C03653=1216.229,222.853,-59.172,-177.266,6.356,148.345
C03654=1216.224,223.101,-59.198,-177.264,6.357,148.345
C03655=1216.220,223.350,-59.222,-177.261,6.359,148.345
C03656=1216.216,223.598,-59.248,-177.259,6.362,148.344
C03657=1216.211,223.848,-59.273,-177.256,6.363,148.344
C03658=1216.206,224.096,-59.298,-177.254,6.365,148.344
C03659=1216.202,224.345,-59.323,-177.251,6.367,148.343
C03660=1216.198,224.593,-59.348,-177.248,6.369,148.343
C03661=1216.193,224.843,-59.373,-177.246,6.371,148.343
C03662=1216.188,225.091,-59.398,-177.243,6.373,148.343
C03663=1216.184,225.340,-59.423,-177.240,6.374,148.342
C03664=1216.179,225.589,-59.449,-177.238,6.377,148.342
C03665=1216.175,225.837,-59.473,-177.236,6.379,148.342
C03666=1216.171,226.086,-59.499,-177.233,6.380,148.341
C03667=1216.166,226.334,-59.524,-177.230,6.382,148.341
C03668=1216.162,226.584,-59.549,-177.228,6.384,148.341
C03669=1216.157,226.832,-59.575,-177.225,6.386,148.340
C03670=1216.152,227.081,-59.600,-177.223,6.388,148.340
C03671=1216.147,227.329,-59.625,-177.220,6.390,148.340
C03672=1216.144,227.578,-59.650,-177.218,6.392,148.340
C03673=1216.139,227.827,-59.675,-177.215,6.394,148.339
C03674=1216.134,228.075,-59.701,-177.212,6.396,148.339
C03675=1216.130,228.324,-59.727,-177.210,6.397,148.339
C03676=1216.125,228.572,-59.752,-177.208,6.400,148.339
C03677=1216.121,228.822,-59.777,-177.205,6.401,148.338
C03678=1216.116,229.070,-59.802,-177.202,6.403,148.338
C03679=1216.112,229.318,-59.828,-177.199,6.406,148.338
C03680=1216.107,229.568,-59.853,-177.197,6.408,148.337
C03681=1216.102,229.816,-59.878,-177.194,6.410,148.337
C03682=1216.098,230.065,-59.904,-177.192,6.412,148.337
C03683=1216.093,230.313,-59.930,-177.189,6.414,148.337
C03684=1216.089,230.562,-59.955,-177.187,6.416,148.336
C03685=1216.085,230.811,-59.980,-177.184,6.417,148.336
C03686=1216.080,231.059,-60.006,-177.181,6.419,148.336
C03687=1216.076,231.308,-60.032,-177.179,6.421,148.336
C03688=1216.071,231.557,-60.057,-177.176,6.423,148.335
C03689=1216.067,231.805,-60.083,-177.174,6.425,148.335
C03690=1216.062,232.054,-60.108,-177.171,6.427,148.335
C03691=1216.058,232.303,-60.133,-177.169,6.429,148.334
C03692=1216.053,232.551,-60.159,-177.166,6.431,148.334
C03693=1216.049,232.800,-60.185,-177.164,6.433,148.334
C03694=1216.045,233.049,-60.210,-177.161,6.435,148.334
C03695=1216.040,233.297,-60.236,-177.159,6.437,148.333
C03696=1216.036,233.546,-60.261,-177.156,6.439,148.333
C03697=1216.031,233.795,-60.287,-177.154,6.441,148.333
C03698=1216.026,234.043,-60.313,-177.151,6.443,148.332
C03699=1216.022,234.292,-60.338,-177.149,6.444,148.332
C03700=1216.018,234.540,-60.364,-177.146,6.446,148.332
C03701=1216.012,234.789,-60.390,-177.143,6.448,148.331
C03702=1216.008,235.038,-60.416,-177.141,6.451,148.331
C03703=1216.004,235.286,-60.442,-177.138,6.453,148.331
C03704=1215.999,235.534,-60.467,-177.135,6.455,148.331
C03705=1215.995,235.783,-60.493,-177.133,6.457,148.330
C03706=1215.991,236.032,-60.518,-177.131,6.459,148.330
C03707=1215.986,236.281,-60.544,-177.128,6.461,148.330
C03708=1215.982,236.529,-60.570,-177.125,6.463,148.330
C03709=1215.977,236.778,-60.596,-177.123,6.464,148.329
C03710=1215.972,237.050,-60.624,-177.120,6.466,148.329
C03711=1215.967,237.321,-60.652,-177.117,6.469,148.329
C03712=1215.962,237.592,-60.680,-177.115,6.471,148.329
C03713=1215.957,237.864,-60.708,-177.112,6.473,148.328
C03714=1215.953,238.112,-60.735,-177.110,6.475,148.328
C03715=1215.949,238.361,-60.760,-177.106,6.478,148.328
C03716=1215.944,238.610,-60.787,-177.104,6.479,148.328
C03717=1215.940,238.859,-60.812,-177.102,6.482,148.327
C03718=1215.935,239.107,-60.838,-177.099,6.484,148.327
C03719=1215.931,239.355,-60.864,-177.096,6.485,148.327
C03720=1215.926,239.604,-60.891,-177.094,6.487,148.326
C03721=1215.922,239.853,-60.916,-177.092,6.489,148.326
C03722=1215.917,240.101,-60.942,-177.089,6.491,148.326
C03723=1215.913,240.350,-60.968,-177.086,6.493,148.326
C03724=1215.908,240.599,-60.994,-177.084,6.495,148.326
C03725=1215.904,240.847,-61.020,-177.082,6.497,148.325
C03726=1215.900,241.096,-61.046,-177.079,6.499,148.325
C03727=1215.895,241.345,-61.072,-177.076,6.502,148.325
C03728=1215.890,241.593,-61.098,-177.074,6.504,148.325
C03729=1215.886,241.841,-61.124,-177.071,6.506,148.324
C03730=1215.882,242.090,-61.150,-177.068,6.508,148.324
C03731=1215.877,242.339,-61.176,-177.066,6.510,148.324
C03732=1215.873,242.587,-61.203,-177.064,6.512,148.324
C03733=1215.869,242.836,-61.229,-177.061,6.514,148.323
C03734=1215.863,243.085,-61.255,-177.058,6.515,148.323
C03735=1215.859,243.333,-61.281,-177.056,6.518,148.323
C03736=1215.854,243.582,-61.307,-177.053,6.520,148.323
C03737=1215.850,243.830,-61.334,-177.050,6.522,148.322
C03738=1215.846,244.079,-61.360,-177.048,6.524,148.322
C03739=1215.841,244.328,-61.386,-177.046,6.526,148.322
C03740=1215.837,244.576,-61.412,-177.043,6.528,148.322
C03741=1215.832,244.824,-61.438,-177.040,6.530,148.321
C03742=1215.828,245.073,-61.465,-177.038,6.532,148.321
C03743=1215.823,245.322,-61.491,-177.036,6.534,148.321
C03744=1215.819,245.570,-61.518,-177.033,6.536,148.321
C03745=1215.815,245.819,-61.543,-177.030,6.539,148.320
C03746=1215.810,246.067,-61.570,-177.028,6.541,148.320
C03747=1215.806,246.316,-61.596,-177.025,6.543,148.320
C03748=1215.802,246.564,-61.623,-177.023,6.545,148.320
C03749=1215.797,246.813,-61.649,-177.020,6.547,148.319
C03750=1215.793,247.062,-61.676,-177.018,6.549,148.319
C03751=1215.788,247.311,-61.702,-177.016,6.551,148.319
C03752=1215.783,247.558,-61.728,-177.013,6.553,148.319
C03753=1215.778,247.807,-61.754,-177.010,6.555,148.318
C03754=1215.774,248.055,-61.781,-177.008,6.557,148.318
C03755=1215.770,248.305,-61.807,-177.005,6.559,148.318
C03756=1215.766,248.553,-61.834,-177.002,6.561,148.318
C03757=1215.761,248.801,-61.861,-177.000,6.563,148.318
C03758=1215.757,249.050,-61.886,-176.998,6.565,148.317
C03759=1215.752,249.299,-61.913,-176.995,6.567,148.317
C03760=1215.747,249.547,-61.941,-176.992,6.570,148.317
C03761=1215.743,249.796,-61.966,-176.990,6.572,148.317
C03762=1215.739,250.044,-61.993,-176.987,6.574,148.316
C03763=1215.735,250.293,-62.020,-176.985,6.576,148.316
C03764=1215.730,250.542,-62.046,-176.982,6.578,148.316
C03765=1215.726,250.790,-62.073,-176.980,6.580,148.316
C03766=1215.721,251.038,-62.100,-176.978,6.582,148.316
C03767=1215.716,251.287,-62.126,-176.974,6.585,148.315
C03768=1215.712,251.536,-62.152,-176.972,6.587,148.315
C03769=1215.708,251.784,-62.180,-176.970,6.589,148.315
C03770=1215.704,252.032,-62.206,-176.967,6.591,148.315
C03771=1215.699,252.281,-62.232,-176.965,6.593,148.315
C03772=1215.694,252.530,-62.259,-176.962,6.595,148.314
C03773=1215.690,252.778,-62.286,-176.959,6.597,148.314
C03774=1215.685,253.027,-62.313,-176.957,6.600,148.314
C03775=1215.681,253.275,-62.340,-176.954,6.601,148.314
C03776=1215.677,253.524,-62.366,-176.952,6.603,148.313
C03777=1215.672,253.772,-62.393,-176.950,6.605,148.313
C03778=1215.667,254.021,-62.420,-176.947,6.607,148.313
C03779=1215.663,254.269,-62.446,-176.944,6.610,148.313
C03780=1215.659,254.518,-62.473,-176.942,6.612,148.312
C03781=1215.654,254.766,-62.500,-176.939,6.614,148.312
C03782=1215.650,255.014,-62.527,-176.937,6.616,148.312
C03783=1215.646,255.263,-62.554,-176.934,6.618,148.312
C03784=1215.641,255.512,-62.581,-176.932,6.621,148.312
C03785=1215.636,255.761,-62.608,-176.929,6.623,148.311
C03786=1215.632,256.009,-62.634,-176.926,6.625,148.311
C03787=1215.628,256.258,-62.661,-176.924,6.627,148.311
C03788=1215.623,256.506,-62.688,-176.922,6.629,148.311
C03789=1215.619,256.755,-62.715,-176.919,6.632,148.311
C03790=1215.615,257.003,-62.742,-176.916,6.634,148.310
C03791=1215.610,257.251,-62.769,-176.914,6.636,148.310
C03792=1215.605,257.500,-62.796,-176.912,6.638,148.310
C03793=1215.601,257.749,-62.823,-176.909,6.640,148.310
C03794=1215.597,257.998,-62.850,-176.906,6.643,148.310
C03795=1215.593,258.246,-62.877,-176.904,6.645,148.309
C03796=1215.588,258.494,-62.904,-176.901,6.647,148.309
C03797=1215.584,258.742,-62.932,-176.899,6.649,148.309
C03798=1215.579,258.991,-62.959,-176.896,6.651,148.309
C03799=1215.574,259.239,-62.986,-176.894,6.654,148.309
C03800=1215.570,259.487,-63.012,-176.891,6.656,148.308
C03801=1215.566,259.737,-63.040,-176.889,6.658,148.308
C03802=1215.562,259.985,-63.067,-176.886,6.660,148.308
C03803=1215.557,260.234,-63.094,-176.884,6.661,148.308
C03804=1215.552,260.482,-63.121,-176.881,6.665,148.308
C03805=1215.548,260.731,-63.148,-176.878,6.666,148.307
C03806=1215.543,260.978,-63.176,-176.876,6.669,148.307
C03807=1215.539,261.228,-63.203,-176.874,6.670,148.307
C03808=1215.535,261.476,-63.230,-176.871,6.673,148.307
C03809=1215.531,261.724,-63.257,-176.868,6.675,148.307
C03810=1215.526,261.973,-63.284,-176.866,6.678,148.306
C03811=1215.522,262.221,-63.312,-176.864,6.679,148.306
C03812=1215.518,262.470,-63.339,-176.861,6.682,148.306
C03813=1215.513,262.718,-63.366,-176.858,6.684,148.306
C03814=1215.508,262.991,-63.396,-176.856,6.686,148.306
C03815=1215.503,263.263,-63.426,-176.853,6.689,148.305
C03816=1215.498,263.536,-63.456,-176.850,6.691,148.305
C03817=1215.494,263.809,-63.487,-176.847,6.694,148.305
C03818=1215.489,264.057,-63.514,-176.845,6.696,148.305
C03819=1215.485,264.306,-63.541,-176.842,6.698,148.305
C03820=1215.480,264.554,-63.568,-176.840,6.701,148.305
C03821=1215.476,264.803,-63.596,-176.837,6.703,148.304
C03822=1215.472,265.051,-63.623,-176.835,6.705,148.304
C03823=1215.467,265.299,-63.651,-176.832,6.707,148.304
C03824=1215.463,265.548,-63.678,-176.830,6.710,148.304
C03825=1215.459,265.797,-63.705,-176.827,6.712,148.303
C03826=1215.454,266.045,-63.733,-176.825,6.714,148.303
C03827=1215.450,266.293,-63.760,-176.822,6.716,148.303
C03828=1215.445,266.541,-63.788,-176.820,6.719,148.303
C03829=1215.440,266.791,-63.816,-176.817,6.721,148.303
C03830=1215.436,267.039,-63.844,-176.815,6.723,148.303
C03831=1215.431,267.287,-63.871,-176.812,6.725,148.302
C03832=1215.428,267.536,-63.899,-176.810,6.728,148.302
C03833=1215.423,267.784,-63.926,-176.807,6.730,148.302
C03834=1215.419,268.032,-63.954,-176.805,6.732,148.302
C03835=1215.414,268.281,-63.981,-176.802,6.734,148.302
C03836=1215.410,268.529,-64.009,-176.800,6.737,148.302
C03837=1215.406,268.778,-64.036,-176.797,6.739,148.301
C03838=1215.401,269.026,-64.064,-176.795,6.741,148.301
C03839=1215.396,269.275,-64.092,-176.792,6.744,148.301
C03840=1215.392,269.523,-64.120,-176.790,6.746,148.301
C03841=1215.387,269.771,-64.147,-176.787,6.748,148.301
C03842=1215.384,270.020,-64.175,-176.785,6.750,148.301
C03843=1215.379,270.268,-64.202,-176.782,6.753,148.300
C03844=1215.374,270.517,-64.230,-176.780,6.755,148.300
C03845=1215.370,270.765,-64.258,-176.777,6.757,148.300
C03846=1215.366,271.014,-64.285,-176.774,6.760,148.300
C03847=1215.362,271.262,-64.313,-176.772,6.762,148.300
C03848=1215.357,271.510,-64.341,-176.769,6.764,148.300
C03849=1215.352,271.759,-64.369,-176.767,6.766,148.299
C03850=1215.348,272.008,-64.397,-176.764,6.769,148.299
C03851=1215.344,272.255,-64.425,-176.762,6.771,148.299
C03852=1215.340,272.503,-64.453,-176.759,6.773,148.299
C03853=1215.335,272.753,-64.481,-176.757,6.776,148.299
C03854=1215.330,273.001,-64.508,-176.755,6.778,148.299
C03855=1215.327,273.249,-64.537,-176.752,6.780,148.298
C03856=1215.322,273.498,-64.564,-176.750,6.782,148.298
C03857=1215.318,273.747,-64.592,-176.747,6.785,148.298
C03858=1215.313,273.995,-64.620,-176.745,6.787,148.298
C03859=1215.309,274.242,-64.648,-176.742,6.789,148.298
C03860=1215.305,274.491,-64.676,-176.739,6.792,148.298
C03861=1215.300,274.740,-64.704,-176.737,6.794,148.298
C03862=1215.296,274.988,-64.732,-176.735,6.796,148.297
C03863=1215.292,275.236,-64.760,-176.732,6.799,148.297
C03864=1215.287,275.485,-64.788,-176.729,6.801,148.297
C03865=1215.283,275.733,-64.816,-176.727,6.803,148.297
C03866=1215.278,275.981,-64.844,-176.724,6.806,148.297
C03867=1215.274,276.230,-64.873,-176.722,6.808,148.297
C03868=1215.269,276.478,-64.900,-176.720,6.810,148.297
C03869=1215.265,276.727,-64.928,-176.717,6.813,148.296
C03870=1215.260,276.975,-64.956,-176.714,6.815,148.296
C03871=1215.257,277.224,-64.984,-176.712,6.817,148.296
C03872=1215.252,277.472,-65.013,-176.709,6.820,148.296
C03873=1215.248,277.720,-65.041,-176.707,6.822,148.296
C03874=1215.243,277.969,-65.069,-176.704,6.824,148.296
C03875=1215.239,278.217,-65.097,-176.702,6.827,148.296
C03876=1215.235,278.465,-65.125,-176.700,6.829,148.295
C03877=1215.230,278.714,-65.154,-176.697,6.831,148.295
C03878=1215.226,278.962,-65.182,-176.694,6.834,148.295
C03879=1215.221,279.211,-65.210,-176.692,6.836,148.295
C03880=1215.217,279.459,-65.238,-176.690,6.838,148.295
C03881=1215.213,279.707,-65.267,-176.687,6.841,148.295
C03882=1215.208,279.955,-65.295,-176.685,6.843,148.295
C03883=1215.204,280.204,-65.323,-176.682,6.845,148.294
C03884=1215.200,280.453,-65.352,-176.680,6.848,148.294
C03885=1215.196,280.700,-65.380,-176.677,6.851,148.294
C03886=1215.191,280.949,-65.409,-176.675,6.852,148.294
C03887=1215.187,281.197,-65.437,-176.672,6.856,148.294
C03888=1215.183,281.446,-65.465,-176.670,6.858,148.294
C03889=1215.177,281.694,-65.494,-176.667,6.860,148.294
C03890=1215.174,281.942,-65.522,-176.665,6.863,148.294
C03891=1215.169,282.191,-65.550,-176.663,6.865,148.294
C03892=1215.165,282.439,-65.579,-176.660,6.867,148.293
C03893=1215.161,282.688,-65.608,-176.657,6.870,148.293
C03894=1215.156,282.935,-65.636,-176.655,6.872,148.293
C03895=1215.152,283.184,-65.664,-176.652,6.875,148.293
C03896=1215.148,283.432,-65.692,-176.650,6.877,148.293
C03897=1215.143,283.680,-65.722,-176.648,6.879,148.293
C03898=1215.139,283.929,-65.750,-176.645,6.882,148.293
C03899=1215.135,284.177,-65.778,-176.642,6.884,148.292
C03900=1215.130,284.426,-65.807,-176.640,6.886,148.292
C03901=1215.125,284.674,-65.836,-176.637,6.889,148.292
C03902=1215.121,284.922,-65.864,-176.635,6.891,148.292
C03903=1215.117,285.171,-65.893,-176.633,6.893,148.292
C03904=1215.113,285.418,-65.921,-176.630,6.896,148.292
C03905=1215.108,285.667,-65.950,-176.628,6.898,148.292
C03906=1215.104,285.916,-65.979,-176.625,6.901,148.292
C03907=1215.100,286.163,-66.007,-176.623,6.903,148.292
C03908=1215.095,286.412,-66.036,-176.620,6.905,148.291
C03909=1215.090,286.660,-66.064,-176.618,6.908,148.291
C03910=1215.087,286.908,-66.093,-176.615,6.911,148.291
C03911=1215.082,287.157,-66.122,-176.613,6.914,148.291
C03912=1215.078,287.405,-66.151,-176.610,6.915,148.291
C03913=1215.073,287.654,-66.180,-176.608,6.918,148.291
C03914=1215.069,287.902,-66.208,-176.605,6.921,148.291
C03915=1215.065,288.151,-66.237,-176.603,6.923,148.291
C03916=1215.060,288.399,-66.266,-176.601,6.925,148.290
C03917=1215.057,288.647,-66.295,-176.598,6.928,148.290
C03918=1215.051,288.921,-66.327,-176.595,6.931,148.290
C03919=1215.046,289.196,-66.358,-176.593,6.933,148.290
C03920=1215.042,289.470,-66.391,-176.590,6.936,148.290
C03921=1215.037,289.744,-66.422,-176.587,6.939,148.290
C03922=1215.033,289.993,-66.451,-176.585,6.941,148.290
C03923=1215.029,290.240,-66.480,-176.582,6.944,148.290
C03924=1215.024,290.488,-66.509,-176.580,6.946,148.290
C03925=1215.020,290.737,-66.538,-176.578,6.948,148.290
C03926=1215.015,290.985,-66.567,-176.575,6.951,148.290
C03927=1215.011,291.234,-66.596,-176.573,6.953,148.289
C03928=1215.007,291.482,-66.625,-176.570,6.956,148.289
C03929=1215.003,291.730,-66.653,-176.568,6.958,148.289
C03930=1214.998,291.978,-66.682,-176.565,6.961,148.289
C03931=1214.994,292.226,-66.712,-176.563,6.964,148.289
C03932=1214.989,292.475,-66.741,-176.560,6.965,148.289
C03933=1214.985,292.723,-66.770,-176.558,6.968,148.289
C03934=1214.981,292.972,-66.800,-176.556,6.971,148.289
C03935=1214.976,293.220,-66.827,-176.553,6.974,148.289
C03936=1214.972,293.468,-66.857,-176.551,6.976,148.289
C03937=1214.968,293.716,-66.886,-176.548,6.978,148.288
C03938=1214.964,293.964,-66.916,-176.545,6.981,148.288
C03939=1214.959,294.213,-66.944,-176.543,6.983,148.288
C03940=1214.955,294.461,-66.973,-176.541,6.986,148.288
C03941=1214.950,294.709,-67.003,-176.539,6.988,148.288
C03942=1214.946,294.957,-67.032,-176.536,6.991,148.288
C03943=1214.942,295.206,-67.061,-176.533,6.993,148.288
C03944=1214.938,295.455,-67.091,-176.531,6.995,148.288
C03945=1214.933,295.702,-67.120,-176.528,6.998,148.288
C03946=1214.929,295.950,-67.149,-176.526,7.001,148.288
C03947=1214.924,296.199,-67.179,-176.524,7.004,148.288
C03948=1214.920,296.447,-67.208,-176.522,7.006,148.288
C03949=1214.916,296.696,-67.237,-176.519,7.009,148.288
C03950=1214.912,296.944,-67.266,-176.516,7.011,148.288
C03951=1214.907,297.192,-67.295,-176.514,7.013,148.287
C03952=1214.903,297.440,-67.325,-176.511,7.016,148.287
C03953=1214.898,297.688,-67.354,-176.509,7.018,148.287
C03954=1214.894,297.936,-67.384,-176.507,7.021,148.287
C03955=1214.890,298.185,-67.413,-176.505,7.024,148.287
C03956=1214.886,298.433,-67.443,-176.502,7.027,148.287
C03957=1214.882,298.681,-67.472,-176.500,7.029,148.287
C03958=1214.878,298.930,-67.501,-176.497,7.032,148.287
C03959=1214.873,299.177,-67.531,-176.495,7.034,148.287
C03960=1214.869,299.425,-67.560,-176.492,7.036,148.287
C03961=1214.864,299.674,-67.589,-176.490,7.039,148.287
C03962=1214.860,299.922,-67.619,-176.488,7.041,148.287
C03963=1214.856,300.170,-67.648,-176.485,7.044,148.287
C03964=1214.852,300.418,-67.678,-176.483,7.046,148.287
C03965=1214.848,300.667,-67.707,-176.480,7.049,148.287
C03966=1214.843,300.915,-67.737,-176.478,7.052,148.287
C03967=1214.839,301.164,-67.767,-176.475,7.055,148.287
C03968=1214.834,301.412,-67.796,-176.473,7.057,148.287
C03969=1214.830,301.660,-67.826,-176.471,7.060,148.287
C03970=1214.825,301.908,-67.855,-176.468,7.062,148.287
C03971=1214.821,302.156,-67.884,-176.466,7.064,148.286
C03972=1214.817,302.404,-67.914,-176.464,7.067,148.286
C03973=1214.812,302.652,-67.944,-176.461,7.070,148.286
C03974=1214.808,302.900,-67.974,-176.459,7.073,148.286
C03975=1214.804,303.149,-68.003,-176.457,7.075,148.286
C03976=1214.800,303.397,-68.033,-176.454,7.078,148.286
C03977=1214.796,303.645,-68.062,-176.451,7.080,148.286
C03978=1214.791,303.894,-68.092,-176.449,7.083,148.286
C03979=1214.787,304.141,-68.122,-176.447,7.085,148.286
C03980=1214.783,304.390,-68.152,-176.444,7.088,148.286
C03981=1214.779,304.638,-68.181,-176.442,7.090,148.286
C03982=1214.774,304.887,-68.211,-176.439,7.093,148.286
C03983=1214.770,305.134,-68.242,-176.437,7.095,148.286
C03984=1214.766,305.382,-68.271,-176.435,7.098,148.286
C03985=1214.761,305.631,-68.301,-176.432,7.101,148.286
C03986=1214.757,305.879,-68.331,-176.430,7.103,148.286
C03987=1214.753,306.127,-68.361,-176.427,7.106,148.286
C03988=1214.748,306.375,-68.390,-176.425,7.108,148.286
C03989=1214.744,306.624,-68.420,-176.423,7.112,148.286
C03990=1214.740,306.871,-68.450,-176.421,7.114,148.286
C03991=1214.735,307.120,-68.480,-176.418,7.117,148.286
C03992=1214.731,307.368,-68.511,-176.416,7.119,148.286
C03993=1214.727,307.616,-68.540,-176.414,7.122,148.286
C03994=1214.723,307.864,-68.570,-176.411,7.124,148.286
C03995=1214.718,308.112,-68.600,-176.409,7.127,148.286
C03996=1214.714,308.360,-68.630,-176.407,7.129,148.286
C03997=1214.710,308.608,-68.660,-176.404,7.133,148.286
C03998=1214.706,308.857,-68.690,-176.402,7.135,148.286
C03999=1214.701,309.106,-68.720,-176.399,7.138,148.286
C04000=1214.697,309.353,-68.750,-176.397,7.140,148.285
C04001=1214.693,309.602,-68.780,-176.394,7.143,148.285
C04002=1214.689,309.849,-68.810,-176.392,7.145,148.285
C04003=1214.684,310.098,-68.840,-176.390,7.148,148.285
C04004=1214.680,310.346,-68.870,-176.387,7.150,148.285
C04005=1214.676,310.594,-68.900,-176.385,7.154,148.286
C04006=1214.671,310.842,-68.931,-176.383,7.156,148.286
C04007=1214.667,311.090,-68.960,-176.381,7.159,148.286
C04008=1214.662,311.338,-68.991,-176.378,7.161,148.285
C04009=1214.659,311.587,-69.021,-176.376,7.164,148.285
C04010=1214.654,311.835,-69.051,-176.374,7.167,148.285
C04011=1214.650,312.083,-69.082,-176.371,7.170,148.285
C04012=1214.645,312.331,-69.112,-176.369,7.172,148.285
C04013=1214.641,312.579,-69.142,-176.367,7.174,148.286
C04014=1214.637,312.827,-69.173,-176.364,7.177,148.286
C04015=1214.633,313.075,-69.202,-176.362,7.180,148.285
C04016=1214.629,313.324,-69.233,-176.360,7.183,148.285
C04017=1214.625,313.571,-69.263,-176.358,7.185,148.285
C04018=1214.620,313.820,-69.293,-176.355,7.188,148.285
C04019=1214.616,314.068,-69.324,-176.353,7.190,148.285
C04020=1214.611,314.316,-69.354,-176.351,7.193,148.286
C04021=1214.607,314.564,-69.384,-176.348,7.196,148.286
C04022=1214.602,314.840,-69.418,-176.346,7.199,148.286
C04023=1214.597,315.116,-69.452,-176.343,7.202,148.286
C04024=1214.593,315.392,-69.486,-176.340,7.205,148.286
C04025=1214.588,315.667,-69.520,-176.338,7.208,148.286
C04026=1214.584,315.917,-69.550,-176.335,7.211,148.286
C04027=1214.580,316.164,-69.580,-176.333,7.213,148.286
C04028=1214.576,316.412,-69.611,-176.331,7.216,148.286
C04029=1214.571,316.660,-69.642,-176.329,7.219,148.286
C04030=1214.567,316.908,-69.672,-176.326,7.222,148.286
C04031=1214.563,317.157,-69.702,-176.324,7.224,148.286
C04032=1214.558,317.405,-69.733,-176.322,7.227,148.286
C04033=1214.554,317.653,-69.763,-176.320,7.229,148.286
C04034=1214.550,317.901,-69.794,-176.317,7.232,148.286
C04035=1214.546,318.149,-69.824,-176.315,7.235,148.286
C04036=1214.542,318.397,-69.855,-176.313,7.238,148.286
C04037=1214.537,318.645,-69.886,-176.311,7.240,148.286
C04038=1214.533,318.893,-69.916,-176.308,7.243,148.286
C04039=1214.529,319.141,-69.947,-176.306,7.245,148.286
C04040=1214.525,319.389,-69.978,-176.304,7.249,148.286
C04041=1214.520,319.637,-70.009,-176.301,7.251,148.286
C04042=1214.516,319.885,-70.038,-176.299,7.254,148.286
C04043=1214.512,320.134,-70.069,-176.297,7.257,148.286
C04044=1214.507,320.382,-70.100,-176.294,7.260,148.286
C04045=1214.503,320.630,-70.130,-176.292,7.262,148.286
C04046=1214.499,320.878,-70.161,-176.290,7.265,148.286
C04047=1214.495,321.126,-70.193,-176.288,7.267,148.286
C04048=1214.491,321.374,-70.224,-176.285,7.270,148.286
C04049=1214.487,321.621,-70.254,-176.283,7.273,148.286
C04050=1214.483,321.870,-70.285,-176.281,7.276,148.286
C04051=1214.478,322.118,-70.316,-176.279,7.278,148.286
C04052=1214.473,322.366,-70.347,-176.276,7.281,148.286
C04053=1214.470,322.614,-70.377,-176.275,7.284,148.287
C04054=1214.466,322.862,-70.408,-176.272,7.287,148.287
C04055=1214.461,323.110,-70.439,-176.270,7.289,148.286
C04056=1214.457,323.359,-70.470,-176.268,7.292,148.287
C04057=1214.452,323.607,-70.500,-176.265,7.295,148.287
C04058=1214.449,323.854,-70.531,-176.263,7.298,148.287
C04059=1214.445,324.102,-70.563,-176.261,7.300,148.287
C04060=1214.440,324.350,-70.593,-176.258,7.303,148.287
C04061=1214.435,324.598,-70.624,-176.257,7.306,148.287
C04062=1214.431,324.847,-70.655,-176.254,7.309,148.287
C04063=1214.427,325.094,-70.687,-176.252,7.311,148.287
C04064=1214.423,325.343,-70.718,-176.250,7.314,148.287
C04065=1214.419,325.591,-70.748,-176.248,7.317,148.287
C04066=1214.415,325.839,-70.779,-176.246,7.320,148.287
C04067=1214.411,326.087,-70.811,-176.243,7.322,148.287
C04068=1214.406,326.335,-70.841,-176.241,7.325,148.288
C04069=1214.402,326.583,-70.872,-176.239,7.328,148.287
C04070=1214.398,326.831,-70.903,-176.236,7.331,148.287
C04071=1214.393,327.079,-70.935,-176.235,7.333,148.288
C04072=1214.389,327.327,-70.966,-176.232,7.336,148.288
C04073=1214.385,327.575,-70.997,-176.230,7.339,148.288
C04074=1214.381,327.823,-71.028,-176.228,7.342,148.288
C04075=1214.376,328.071,-71.059,-176.226,7.344,148.288
C04076=1214.372,328.319,-71.090,-176.224,7.347,148.288
C04077=1214.368,328.567,-71.122,-176.222,7.350,148.288
C04078=1214.364,328.815,-71.153,-176.219,7.353,148.288
C04079=1214.361,329.063,-71.184,-176.217,7.356,148.288
C04080=1214.356,329.311,-71.215,-176.215,7.358,148.288
C04081=1214.352,329.560,-71.246,-176.213,7.362,148.289
C04082=1214.348,329.807,-71.277,-176.211,7.364,148.289
C04083=1214.343,330.056,-71.309,-176.208,7.367,148.289
C04084=1214.339,330.303,-71.340,-176.206,7.370,148.289
C04085=1214.334,330.551,-71.371,-176.204,7.373,148.289
C04086=1214.330,330.799,-71.403,-176.202,7.375,148.289
C04087=1214.326,331.047,-71.434,-176.200,7.379,148.289
C04088=1214.322,331.295,-71.466,-176.198,7.381,148.289
C04089=1214.317,331.543,-71.496,-176.195,7.384,148.289
C04090=1214.314,331.791,-71.528,-176.193,7.386,148.289
C04091=1214.309,332.039,-71.559,-176.191,7.390,148.289
C04092=1214.305,332.287,-71.591,-176.189,7.392,148.290
C04093=1214.301,332.535,-71.622,-176.187,7.395,148.290
C04094=1214.297,332.783,-71.653,-176.185,7.398,148.290
C04095=1214.293,333.030,-71.685,-176.183,7.401,148.290
C04096=1214.289,333.279,-71.716,-176.181,7.403,148.290
C04097=1214.284,333.527,-71.748,-176.178,7.406,148.290
C04098=1214.280,333.775,-71.779,-176.177,7.409,148.290
C04099=1214.275,334.023,-71.811,-176.174,7.412,148.290
C04100=1214.272,334.271,-71.843,-176.172,7.414,148.290
C04101=1214.267,334.519,-71.873,-176.170,7.418,148.291
C04102=1214.263,334.767,-71.905,-176.168,7.420,148.291
C04103=1214.260,335.015,-71.937,-176.166,7.423,148.291
C04104=1214.254,335.263,-71.968,-176.164,7.426,148.291
C04105=1214.250,335.511,-72.000,-176.162,7.429,148.291
C04106=1214.246,335.759,-72.032,-176.160,7.431,148.291
C04107=1214.242,336.007,-72.064,-176.158,7.435,148.291
C04108=1214.238,336.255,-72.094,-176.156,7.437,148.292
C04109=1214.233,336.503,-72.127,-176.153,7.440,148.292
C04110=1214.229,336.750,-72.158,-176.152,7.443,148.292
C04111=1214.225,336.998,-72.190,-176.149,7.446,148.292
C04112=1214.221,337.247,-72.221,-176.147,7.448,148.292
C04113=1214.217,337.494,-72.253,-176.145,7.452,148.292
C04114=1214.213,337.743,-72.285,-176.143,7.454,148.292
C04115=1214.208,337.990,-72.317,-176.141,7.457,148.292
C04116=1214.205,338.238,-72.348,-176.139,7.460,148.292
C04117=1214.201,338.487,-72.380,-176.137,7.463,148.293
C04118=1214.196,338.734,-72.412,-176.135,7.466,148.293
C04119=1214.192,338.982,-72.444,-176.133,7.469,148.293
C04120=1214.188,339.230,-72.475,-176.131,7.471,148.293
C04121=1214.183,339.478,-72.507,-176.129,7.475,148.293
C04122=1214.179,339.726,-72.539,-176.127,7.477,148.293
C04123=1214.175,339.973,-72.571,-176.124,7.480,148.293
C04124=1214.171,340.221,-72.603,-176.123,7.483,148.294
C04125=1214.167,340.470,-72.635,-176.121,7.486,148.294
C04126=1214.162,340.748,-72.670,-176.118,7.489,148.294
C04127=1214.157,341.026,-72.706,-176.117,7.492,148.294
C04128=1214.153,341.303,-72.742,-176.114,7.495,148.294
C04129=1214.148,341.582,-72.777,-176.112,7.498,148.295
C04130=1214.144,341.830,-72.809,-176.110,7.502,148.295
C04131=1214.139,342.078,-72.842,-176.108,7.504,148.295
C04132=1214.135,342.325,-72.873,-176.106,7.508,148.295
C04133=1214.131,342.574,-72.905,-176.104,7.510,148.295
C04134=1214.127,342.821,-72.938,-176.102,7.513,148.295
C04135=1214.123,343.069,-72.969,-176.100,7.516,148.296
C04136=1214.119,343.317,-73.002,-176.098,7.519,148.296
C04137=1214.115,343.565,-73.034,-176.096,7.522,148.296
C04138=1214.110,343.813,-73.066,-176.094,7.525,148.296
C04139=1214.106,344.061,-73.098,-176.092,7.527,148.296
C04140=1214.102,344.309,-73.130,-176.090,7.531,148.297
C04141=1214.097,344.556,-73.162,-176.088,7.533,148.297
C04142=1214.094,344.804,-73.193,-176.086,7.536,148.297
C04143=1214.089,345.053,-73.226,-176.084,7.539,148.297
C04144=1214.085,345.301,-73.258,-176.082,7.542,148.297
C04145=1214.081,345.548,-73.291,-176.080,7.545,148.297
C04146=1214.077,345.796,-73.322,-176.079,7.547,148.298
C04147=1214.073,346.044,-73.355,-176.076,7.551,148.298
C04148=1214.068,346.292,-73.386,-176.075,7.553,148.298
C04149=1214.064,346.540,-73.419,-176.073,7.556,148.298
C04150=1214.060,346.787,-73.451,-176.071,7.559,148.298
C04151=1214.056,347.036,-73.484,-176.069,7.562,148.299
C04152=1214.052,347.283,-73.515,-176.067,7.565,148.299
C04153=1214.047,347.531,-73.548,-176.065,7.568,148.299
C04154=1214.044,347.779,-73.580,-176.063,7.571,148.299
C04155=1214.039,348.027,-73.613,-176.061,7.574,148.299
C04156=1214.036,348.275,-73.644,-176.059,7.577,148.300
C04157=1214.031,348.523,-73.677,-176.057,7.580,148.300
C04158=1214.026,348.771,-73.710,-176.055,7.582,148.300
C04159=1214.023,349.019,-73.742,-176.054,7.585,148.300
C04160=1214.018,349.267,-73.774,-176.052,7.588,148.300
C04161=1214.014,349.514,-73.806,-176.050,7.591,148.301
C04162=1214.010,349.762,-73.839,-176.048,7.594,148.301
C04163=1214.005,350.010,-73.871,-176.046,7.597,148.301
C04164=1214.002,350.258,-73.904,-176.044,7.600,148.301
C04165=1213.998,350.506,-73.936,-176.043,7.603,148.302
C04166=1213.994,350.753,-73.968,-176.041,7.606,148.302
C04167=1213.989,351.001,-74.001,-176.039,7.609,148.302
C04168=1213.985,351.250,-74.033,-176.037,7.612,148.302
C04169=1213.981,351.497,-74.066,-176.035,7.615,148.302
C04170=1213.977,351.745,-74.098,-176.033,7.617,148.303
C04171=1213.973,351.993,-74.131,-176.031,7.620,148.303
C04172=1213.968,352.240,-74.163,-176.030,7.623,148.303
C04173=1213.964,352.488,-74.196,-176.028,7.627,148.303
C04174=1213.960,352.736,-74.228,-176.026,7.629,148.304
C04175=1213.956,352.984,-74.261,-176.024,7.633,148.304
C04176=1213.952,353.232,-74.293,-176.022,7.635,148.304
C04177=1213.948,353.480,-74.327,-176.021,7.638,148.304
C04178=1213.944,353.727,-74.358,-176.019,7.641,148.305
C04179=1213.939,353.975,-74.391,-176.017,7.644,148.305
C04180=1213.935,354.223,-74.424,-176.015,7.647,148.305
C04181=1213.931,354.471,-74.457,-176.013,7.650,148.305
C04182=1213.927,354.719,-74.489,-176.011,7.653,148.305
C04183=1213.923,354.967,-74.522,-176.010,7.656,148.306
C04184=1213.919,355.215,-74.555,-176.008,7.658,148.306
C04185=1213.915,355.463,-74.587,-176.006,7.662,148.306
C04186=1213.911,355.710,-74.620,-176.005,7.664,148.306
C04187=1213.906,355.958,-74.652,-176.003,7.668,148.307
C04188=1213.902,356.206,-74.685,-176.001,7.670,148.307
C04189=1213.898,356.453,-74.718,-176.000,7.673,148.307
C04190=1213.894,356.701,-74.750,-175.998,7.676,148.308
C04191=1213.890,356.949,-74.783,-175.996,7.679,148.308
C04192=1213.886,357.197,-74.816,-175.994,7.682,148.308
C04193=1213.881,357.445,-74.849,-175.993,7.685,148.309
C04194=1213.878,357.693,-74.881,-175.991,7.688,148.309
C04195=1213.874,357.940,-74.915,-175.989,7.691,148.309
C04196=1213.870,358.188,-74.948,-175.988,7.694,148.309
C04197=1213.865,358.437,-74.980,-175.986,7.697,148.310
C04198=1213.861,358.684,-75.013,-175.984,7.700,148.310
C04199=1213.857,358.932,-75.047,-175.983,7.703,148.310
C04200=1213.853,359.179,-75.079,-175.980,7.706,148.310
C04201=1213.848,359.427,-75.111,-175.979,7.709,148.311
C04202=1213.844,359.675,-75.144,-175.977,7.712,148.311
C04203=1213.840,359.923,-75.177,-175.975,7.715,148.311
C04204=1213.836,360.170,-75.211,-175.974,7.717,148.312
C04205=1213.832,360.418,-75.244,-175.972,7.721,148.312
C04206=1213.827,360.666,-75.276,-175.971,7.724,148.312
C04207=1213.823,360.914,-75.309,-175.969,7.726,148.312
C04208=1213.820,361.161,-75.342,-175.967,7.730,148.313
C04209=1213.816,361.409,-75.375,-175.966,7.732,148.313
C04210=1213.812,361.657,-75.408,-175.965,7.735,148.313
C04211=1213.807,361.905,-75.441,-175.962,7.738,148.314
C04212=1213.803,362.152,-75.475,-175.961,7.741,148.314
C04213=1213.799,362.401,-75.507,-175.960,7.744,148.314
C04214=1213.795,362.648,-75.540,-175.958,7.747,148.315
C04215=1213.791,362.896,-75.573,-175.956,7.750,148.315
C04216=1213.786,363.144,-75.606,-175.955,7.753,148.315
C04217=1213.782,363.392,-75.640,-175.953,7.756,148.315
C04218=1213.778,363.639,-75.673,-175.952,7.759,148.316
C04219=1213.774,363.887,-75.706,-175.950,7.761,148.316
C04220=1213.770,364.135,-75.739,-175.948,7.765,148.316
C04221=1213.766,364.383,-75.772,-175.947,7.768,148.317
C04222=1213.762,364.631,-75.806,-175.945,7.770,148.317
C04223=1213.758,364.879,-75.839,-175.944,7.774,148.317
C04224=1213.754,365.126,-75.872,-175.942,7.777,148.318
C04225=1213.750,365.374,-75.905,-175.941,7.779,148.318
C04226=1213.746,365.622,-75.938,-175.940,7.782,148.318
C04227=1213.742,365.870,-75.972,-175.937,7.786,148.319
C04228=1213.737,366.117,-76.005,-175.936,7.788,148.319
C04229=1213.733,366.365,-76.038,-175.935,7.791,148.319
C04230=1213.729,366.645,-76.075,-175.933,7.795,148.320
C04231=1213.725,366.925,-76.113,-175.931,7.798,148.320
C04232=1213.719,367.206,-76.151,-175.930,7.801,148.321
C04233=1213.715,367.486,-76.189,-175.928,7.805,148.321
C04234=1213.711,367.734,-76.222,-175.927,7.807,148.321
C04235=1213.707,367.981,-76.255,-175.925,7.810,148.322
C04236=1213.703,368.229,-76.288,-175.924,7.814,148.322
C04237=1213.699,368.476,-76.322,-175.922,7.816,148.322
C04238=1213.695,368.724,-76.355,-175.921,7.819,148.323
C04239=1213.691,368.972,-76.388,-175.920,7.822,148.323
C04240=1213.686,369.219,-76.421,-175.918,7.825,148.323
C04241=1213.682,369.467,-76.455,-175.917,7.828,148.324
C04242=1213.677,369.715,-76.488,-175.915,7.831,148.324
C04243=1213.674,369.963,-76.523,-175.914,7.834,148.325
C04244=1213.670,370.211,-76.556,-175.913,7.837,148.325
C04245=1213.666,370.458,-76.589,-175.911,7.839,148.325
C04246=1213.662,370.706,-76.622,-175.910,7.843,148.326
C04247=1213.658,370.953,-76.656,-175.908,7.846,148.326
C04248=1213.653,371.201,-76.690,-175.907,7.848,148.326
C04249=1213.649,371.449,-76.723,-175.906,7.851,148.327
C04250=1213.645,371.697,-76.756,-175.905,7.854,148.327
C04251=1213.642,371.944,-76.790,-175.904,7.857,148.328
C04252=1213.637,372.192,-76.823,-175.902,7.860,148.328
C04253=1213.633,372.440,-76.857,-175.901,7.863,148.328
C04254=1213.628,372.688,-76.890,-175.900,7.866,148.329
C04255=1213.625,372.935,-76.924,-175.898,7.869,148.329
C04256=1213.620,373.183,-76.957,-175.897,7.872,148.329
C04257=1213.616,373.431,-76.990,-175.895,7.874,148.330
C04258=1213.613,373.678,-77.025,-175.894,7.877,148.330
C04259=1213.608,373.926,-77.058,-175.893,7.880,148.331
C04260=1213.604,374.173,-77.092,-175.892,7.883,148.331
C04261=1213.600,374.421,-77.125,-175.891,7.886,148.331
C04262=1213.596,374.669,-77.159,-175.890,7.888,148.332
C04263=1213.592,374.917,-77.193,-175.888,7.892,148.332
C04264=1213.588,375.165,-77.227,-175.887,7.895,148.333
C04265=1213.584,375.413,-77.260,-175.885,7.898,148.333
C04266=1213.580,375.660,-77.294,-175.884,7.901,148.333
C04267=1213.575,375.908,-77.327,-175.883,7.903,148.334
C04268=1213.572,376.155,-77.362,-175.882,7.906,148.334
C04269=1213.568,376.403,-77.395,-175.881,7.909,148.335
C04270=1213.564,376.650,-77.429,-175.880,7.912,148.335
C04271=1213.559,376.898,-77.462,-175.879,7.915,148.336
C04272=1213.555,377.145,-77.496,-175.877,7.918,148.336
C04273=1213.552,377.394,-77.530,-175.876,7.921,148.336
C04274=1213.547,377.641,-77.564,-175.875,7.923,148.337
C04275=1213.543,377.889,-77.597,-175.874,7.926,148.337
C04276=1213.539,378.137,-77.631,-175.873,7.929,148.338
C04277=1213.534,378.384,-77.665,-175.872,7.932,148.338
C04278=1213.531,378.632,-77.699,-175.871,7.935,148.339
C04279=1213.527,378.880,-77.732,-175.870,7.938,148.339
C04280=1213.522,379.127,-77.767,-175.868,7.941,148.339
C04281=1213.518,379.375,-77.800,-175.867,7.943,148.340
C04282=1213.515,379.623,-77.834,-175.867,7.945,148.340
C04283=1213.510,379.871,-77.868,-175.866,7.948,148.341
C04284=1213.506,380.118,-77.902,-175.865,7.951,148.341
C04285=1213.502,380.366,-77.935,-175.863,7.954,148.341
C04286=1213.498,380.614,-77.970,-175.862,7.957,148.342
C04287=1213.494,380.861,-78.004,-175.861,7.960,148.342
C04288=1213.489,381.109,-78.038,-175.860,7.963,148.343
C04289=1213.486,381.356,-78.071,-175.859,7.966,148.343
C04290=1213.482,381.604,-78.105,-175.858,7.968,148.344
C04291=1213.477,381.852,-78.139,-175.857,7.971,148.344
C04292=1213.474,382.099,-78.173,-175.856,7.974,148.345
C04293=1213.469,382.347,-78.207,-175.855,7.976,148.345
C04294=1213.466,382.595,-78.241,-175.854,7.979,148.345
C04295=1213.462,382.842,-78.275,-175.853,7.982,148.346
C04296=1213.457,383.090,-78.309,-175.852,7.985,148.346
C04297=1213.454,383.338,-78.343,-175.851,7.988,148.347
C04298=1213.449,383.585,-78.378,-175.850,7.990,148.347
C04299=1213.445,383.833,-78.411,-175.850,7.993,148.348
C04300=1213.440,384.080,-78.445,-175.848,7.996,148.348
C04301=1213.437,384.328,-78.479,-175.847,7.999,148.348
C04302=1213.432,384.576,-78.513,-175.846,8.002,148.349
C04303=1213.428,384.823,-78.547,-175.846,8.004,148.349
C04304=1213.425,385.071,-78.581,-175.845,8.006,148.350
C04305=1213.421,385.318,-78.616,-175.844,8.010,148.350
C04306=1213.416,385.566,-78.649,-175.843,8.012,148.351
C04307=1213.412,385.814,-78.684,-175.842,8.016,148.351
C04308=1213.409,386.061,-78.718,-175.841,8.017,148.352
C04309=1213.404,386.309,-78.752,-175.840,8.020,148.352
C04310=1213.401,386.557,-78.786,-175.839,8.023,148.353
C04311=1213.396,386.805,-78.820,-175.838,8.026,148.353
C04312=1213.392,387.052,-78.854,-175.837,8.028,148.353
C04313=1213.388,387.300,-78.889,-175.837,8.031,148.354
C04314=1213.384,387.547,-78.923,-175.836,8.034,148.354
C04315=1213.380,387.794,-78.957,-175.835,8.036,148.355
C04316=1213.376,388.043,-78.991,-175.834,8.039,148.355
C04317=1213.372,388.290,-79.025,-175.833,8.042,148.356
C04318=1213.368,388.537,-79.059,-175.833,8.044,148.356
C04319=1213.364,388.786,-79.094,-175.832,8.047,148.357
C04320=1213.359,389.033,-79.128,-175.831,8.050,148.357
C04321=1213.355,389.280,-79.162,-175.830,8.052,148.358
C04322=1213.351,389.529,-79.196,-175.829,8.055,148.358
C04323=1213.347,389.776,-79.230,-175.828,8.058,148.359
C04324=1213.343,390.023,-79.265,-175.828,8.060,148.359
C04325=1213.340,390.271,-79.299,-175.827,8.063,148.360
C04326=1213.335,390.519,-79.333,-175.826,8.066,148.360
C04327=1213.332,390.766,-79.368,-175.825,8.068,148.360
C04328=1213.327,391.014,-79.402,-175.825,8.071,148.361
C04329=1213.323,391.261,-79.436,-175.824,8.073,148.361
C04330=1213.319,391.509,-79.471,-175.823,8.076,148.362
C04331=1213.315,391.756,-79.505,-175.822,8.079,148.362
C04332=1213.312,392.004,-79.539,-175.822,8.082,148.363
C04333=1213.307,392.252,-79.574,-175.821,8.084,148.363
C04334=1213.302,392.534,-79.613,-175.820,8.087,148.364
C04335=1213.298,392.816,-79.652,-175.820,8.090,148.364
C04336=1213.293,393.098,-79.691,-175.818,8.093,148.365
C04337=1213.289,393.381,-79.730,-175.818,8.096,148.365
C04338=1213.284,393.628,-79.765,-175.817,8.099,148.366
C04339=1213.280,393.875,-79.799,-175.816,8.101,148.366
C04340=1213.276,394.123,-79.834,-175.816,8.104,148.367
C04341=1213.272,394.371,-79.868,-175.815,8.106,148.367
C04342=1213.269,394.618,-79.902,-175.814,8.109,148.368
C04343=1213.264,394.866,-79.937,-175.814,8.111,148.368
C04344=1213.260,395.113,-79.971,-175.813,8.114,148.369
C04345=1213.256,395.361,-80.005,-175.812,8.116,148.369
C04346=1213.252,395.609,-80.040,-175.811,8.119,148.370
C04347=1213.248,395.856,-80.074,-175.811,8.121,148.370
C04348=1213.244,396.104,-80.109,-175.810,8.124,148.371
C04349=1213.240,396.352,-80.143,-175.810,8.126,148.371
C04350=1213.235,396.599,-80.178,-175.809,8.129,148.372
C04351=1213.232,396.846,-80.212,-175.808,8.132,148.372
C04352=1213.228,397.095,-80.247,-175.808,8.134,148.373
C04353=1213.223,397.342,-80.281,-175.807,8.137,148.373
C04354=1213.220,397.590,-80.315,-175.806,8.139,148.373
C04355=1213.215,397.837,-80.351,-175.806,8.142,148.374
C04356=1213.212,398.085,-80.385,-175.805,8.144,148.375
C04357=1213.208,398.332,-80.419,-175.805,8.146,148.375
C04358=1213.204,398.580,-80.454,-175.804,8.149,148.376
C04359=1213.199,398.827,-80.489,-175.803,8.151,148.376
C04360=1213.195,399.075,-80.523,-175.803,8.154,148.376
C04361=1213.191,399.323,-80.557,-175.802,8.156,148.377
C04362=1213.187,399.570,-80.592,-175.802,8.158,148.377
C04363=1213.183,399.817,-80.627,-175.801,8.162,148.378
C04364=1213.179,400.065,-80.661,-175.800,8.163,148.378
C04365=1213.175,400.313,-80.696,-175.800,8.166,148.379
C04366=1213.171,400.560,-80.730,-175.799,8.169,148.379
C04367=1213.167,400.808,-80.765,-175.799,8.171,148.380
C04368=1213.163,401.055,-80.799,-175.799,8.173,148.380
C04369=1213.159,401.303,-80.835,-175.797,8.176,148.381
C04370=1213.155,401.550,-80.869,-175.797,8.178,148.381
C04371=1213.151,401.798,-80.904,-175.796,8.180,148.382
C04372=1213.147,402.046,-80.938,-175.796,8.182,148.382
C04373=1213.143,402.294,-80.973,-175.796,8.186,148.383
C04374=1213.139,402.540,-81.008,-175.795,8.188,148.383
C04375=1213.135,402.789,-81.043,-175.795,8.190,148.384
C04376=1213.130,403.036,-81.077,-175.793,8.193,148.384
C04377=1213.127,403.284,-81.111,-175.793,8.195,148.384
C04378=1213.123,403.531,-81.147,-175.793,8.197,148.385
C04379=1213.119,403.779,-81.181,-175.792,8.199,148.385
C04380=1213.114,404.026,-81.216,-175.792,8.202,148.386
C04381=1213.111,404.274,-81.250,-175.791,8.204,148.386
C04382=1213.107,404.521,-81.285,-175.791,8.206,148.387
C04383=1213.103,404.769,-81.320,-175.791,8.209,148.387
C04384=1213.098,405.016,-81.355,-175.790,8.211,148.388
C04385=1213.094,405.264,-81.389,-175.789,8.214,148.388
C04386=1213.091,405.511,-81.424,-175.789,8.216,148.389
C04387=1213.087,405.759,-81.459,-175.788,8.218,148.389
C04388=1213.082,406.006,-81.493,-175.788,8.220,148.390
C04389=1213.078,406.254,-81.529,-175.787,8.222,148.390
C04390=1213.074,406.501,-81.563,-175.787,8.225,148.391
C04391=1213.070,406.749,-81.598,-175.786,8.227,148.391
C04392=1213.066,406.996,-81.633,-175.786,8.230,148.391
C04393=1213.062,407.244,-81.668,-175.786,8.232,148.392
C04394=1213.058,407.491,-81.702,-175.785,8.234,148.392
C04395=1213.054,407.739,-81.738,-175.785,8.236,148.393
C04396=1213.050,407.986,-81.772,-175.784,8.239,148.393
C04397=1213.046,408.235,-81.807,-175.783,8.241,148.394
C04398=1213.041,408.481,-81.842,-175.783,8.244,148.394
C04399=1213.038,408.729,-81.876,-175.782,8.245,148.395
C04400=1213.034,408.977,-81.911,-175.782,8.248,148.395
C04401=1213.030,409.224,-81.946,-175.782,8.250,148.396
C04402=1213.026,409.472,-81.981,-175.781,8.252,148.396
C04403=1213.022,409.719,-82.016,-175.781,8.255,148.397
C04404=1213.018,409.967,-82.051,-175.780,8.257,148.397
C04405=1213.013,410.215,-82.086,-175.780,8.259,148.398
C04406=1213.010,410.462,-82.121,-175.779,8.261,148.398
C04407=1213.006,410.709,-82.155,-175.779,8.264,148.398
C04408=1213.002,410.957,-82.191,-175.779,8.266,148.399
C04409=1212.998,411.205,-82.225,-175.778,8.268,148.399
C04410=1212.993,411.452,-82.260,-175.778,8.270,148.400
C04411=1212.990,411.700,-82.295,-175.777,8.272,148.400
C04412=1212.985,411.947,-82.330,-175.777,8.274,148.401
C04413=1212.981,412.195,-82.365,-175.777,8.277,148.401
C04414=1212.977,412.442,-82.400,-175.776,8.279,148.402
C04415=1212.973,412.690,-82.435,-175.776,8.281,148.402
C04416=1212.970,412.937,-82.470,-175.775,8.284,148.403
C04417=1212.966,413.184,-82.505,-175.775,8.286,148.403
C04418=1212.962,413.432,-82.540,-175.774,8.288,148.403
C04419=1212.958,413.679,-82.575,-175.774,8.290,148.404
C04420=1212.954,413.927,-82.610,-175.773,8.292,148.404
C04421=1212.949,414.174,-82.645,-175.773,8.294,148.405
C04422=1212.945,414.422,-82.680,-175.773,8.297,148.405
C04423=1212.942,414.670,-82.715,-175.772,8.299,148.406
C04424=1212.937,414.917,-82.750,-175.772,8.301,148.406
C04425=1212.933,415.165,-82.785,-175.771,8.303,148.407
C04426=1212.929,415.405,-82.819,-175.771,8.305,148.407
C04427=1212.926,415.646,-82.853,-175.770,8.307,148.407
C04428=1212.921,415.887,-82.887,-175.770,8.309,148.408
C04429=1212.917,416.128,-82.921,-175.769,8.311,148.408
C04430=1212.914,416.369,-82.956,-175.770,8.313,148.409
C04431=1212.910,416.609,-82.989,-175.769,8.315,148.409
C04432=1212.908,416.851,-83.023,-175.769,8.317,148.410
C04433=1212.909,417.091,-83.057,-175.768,8.319,148.410
C04434=1212.488,417.091,-83.093,-175.771,8.330,148.414
C04435=1212.487,416.850,-83.059,-175.772,8.328,148.413
C04436=1212.488,416.607,-83.025,-175.772,8.325,148.413
C04437=1212.492,416.365,-82.991,-175.772,8.324,148.413
C04438=1212.495,416.122,-82.957,-175.773,8.322,148.412
C04439=1212.500,415.881,-82.922,-175.773,8.320,148.412
C04440=1212.504,415.638,-82.888,-175.774,8.318,148.411
C04441=1212.507,415.397,-82.854,-175.774,8.316,148.411
C04442=1212.511,415.154,-82.819,-175.774,8.314,148.410
C04443=1212.516,414.907,-82.785,-175.775,8.311,148.410
C04444=1212.519,414.659,-82.749,-175.775,8.309,148.409
C04445=1212.523,414.411,-82.714,-175.775,8.307,148.409
C04446=1212.528,414.164,-82.679,-175.776,8.305,148.409
C04447=1212.532,413.916,-82.644,-175.776,8.303,148.408
C04448=1212.536,413.669,-82.609,-175.777,8.301,148.408
C04449=1212.540,413.421,-82.574,-175.777,8.299,148.407
C04450=1212.544,413.174,-82.539,-175.777,8.296,148.407
C04451=1212.548,412.926,-82.504,-175.778,8.294,148.406
C04452=1212.552,412.679,-82.469,-175.779,8.291,148.406
C04453=1212.556,412.431,-82.434,-175.779,8.289,148.405
C04454=1212.559,412.184,-82.399,-175.780,8.287,148.405
C04455=1212.564,411.937,-82.365,-175.780,8.285,148.404
C04456=1212.567,411.689,-82.329,-175.781,8.283,148.404
C04457=1212.571,411.441,-82.295,-175.781,8.280,148.403
C04458=1212.576,411.194,-82.259,-175.781,8.278,148.403
C04459=1212.580,410.946,-82.225,-175.782,8.276,148.403
C04460=1212.584,410.699,-82.190,-175.782,8.274,148.402
C04461=1212.588,410.451,-82.155,-175.782,8.272,148.402
C04462=1212.592,410.204,-82.120,-175.783,8.270,148.401
C04463=1212.596,409.956,-82.085,-175.783,8.268,148.401
C04464=1212.599,409.708,-82.050,-175.784,8.265,148.400
C04465=1212.604,409.461,-82.016,-175.785,8.263,148.400
C04466=1212.608,409.214,-81.980,-175.785,8.260,148.399
C04467=1212.612,408.966,-81.946,-175.785,8.258,148.399
C04468=1212.616,408.719,-81.910,-175.786,8.256,148.398
C04469=1212.620,408.471,-81.876,-175.786,8.254,148.398
C04470=1212.624,408.223,-81.841,-175.787,8.252,148.398
C04471=1212.628,407.977,-81.806,-175.787,8.250,148.397
C04472=1212.632,407.728,-81.772,-175.787,8.247,148.396
C04473=1212.636,407.480,-81.737,-175.788,8.245,148.396
C04474=1212.640,407.234,-81.702,-175.789,8.242,148.396
C04475=1212.644,406.985,-81.667,-175.789,8.240,148.395
C04476=1212.649,406.738,-81.632,-175.789,8.238,148.395
C04477=1212.652,406.491,-81.597,-175.790,8.236,148.394
C04478=1212.656,406.243,-81.563,-175.790,8.234,148.394
C04479=1212.660,405.995,-81.528,-175.791,8.231,148.393
C04480=1212.664,405.748,-81.493,-175.791,8.228,148.393
C04481=1212.668,405.500,-81.458,-175.792,8.226,148.392
C04482=1212.673,405.253,-81.423,-175.792,8.224,148.392
C04483=1212.676,405.006,-81.389,-175.793,8.222,148.391
C04484=1212.680,404.758,-81.354,-175.793,8.219,148.391
C04485=1212.684,404.510,-81.319,-175.794,8.217,148.390
C04486=1212.689,404.263,-81.285,-175.794,8.215,148.390
C04487=1212.693,404.015,-81.249,-175.795,8.213,148.389
C04488=1212.697,403.768,-81.215,-175.795,8.209,148.389
C04489=1212.700,403.520,-81.181,-175.796,8.207,148.389
C04490=1212.705,403.273,-81.145,-175.796,8.205,148.388
C04491=1212.709,403.025,-81.110,-175.797,8.203,148.388
C04492=1212.713,402.778,-81.076,-175.798,8.200,148.387
C04493=1212.716,402.530,-81.042,-175.798,8.198,148.387
C04494=1212.721,402.283,-81.007,-175.798,8.196,148.386
C04495=1212.725,402.035,-80.972,-175.799,8.194,148.386
C04496=1212.729,401.788,-80.937,-175.800,8.191,148.385
C04497=1212.733,401.539,-80.902,-175.800,8.189,148.385
C04498=1212.737,401.292,-80.869,-175.800,8.186,148.384
C04499=1212.741,401.045,-80.833,-175.801,8.183,148.384
C04500=1212.745,400.797,-80.799,-175.802,8.181,148.383
C04501=1212.749,400.549,-80.764,-175.802,8.179,148.383
C04502=1212.753,400.302,-80.730,-175.803,8.176,148.382
C04503=1212.757,400.054,-80.695,-175.803,8.174,148.382
C04504=1212.762,399.807,-80.661,-175.804,8.172,148.381
C04505=1212.765,399.559,-80.625,-175.805,8.169,148.381
C04506=1212.769,399.312,-80.591,-175.805,8.167,148.381
C04507=1212.774,399.065,-80.557,-175.806,8.165,148.380
C04508=1212.778,398.817,-80.522,-175.806,8.161,148.379
C04509=1212.781,398.569,-80.488,-175.807,8.159,148.379
C04510=1212.785,398.321,-80.453,-175.807,8.157,148.379
C04511=1212.790,398.074,-80.419,-175.808,8.154,148.378
C04512=1212.794,397.826,-80.383,-175.809,8.152,148.378
C04513=1212.797,397.579,-80.349,-175.809,8.149,148.377
C04514=1212.801,397.331,-80.314,-175.810,8.147,148.377
C04515=1212.806,397.084,-80.280,-175.810,8.145,148.376
C04516=1212.809,396.836,-80.246,-175.811,8.142,148.376
C04517=1212.814,396.588,-80.211,-175.812,8.140,148.375
C04518=1212.818,396.341,-80.177,-175.813,8.137,148.375
C04519=1212.822,396.093,-80.143,-175.813,8.135,148.374
C04520=1212.826,395.846,-80.108,-175.814,8.131,148.374
C04521=1212.830,395.598,-80.073,-175.814,8.129,148.373
C04522=1212.834,395.351,-80.039,-175.815,8.126,148.373
C04523=1212.838,395.102,-80.005,-175.816,8.124,148.372
C04524=1212.842,394.856,-79.969,-175.816,8.121,148.372
C04525=1212.846,394.609,-79.936,-175.817,8.119,148.371
C04526=1212.850,394.360,-79.901,-175.817,8.117,148.371
C04527=1212.855,394.113,-79.866,-175.818,8.114,148.370
C04528=1212.858,393.865,-79.832,-175.819,8.111,148.370
C04529=1212.862,393.618,-79.798,-175.819,8.109,148.369
C04530=1212.867,393.370,-79.763,-175.821,8.106,148.369
C04531=1212.871,393.088,-79.725,-175.821,8.104,148.368
C04532=1212.876,392.806,-79.685,-175.822,8.101,148.368
C04533=1212.880,392.523,-79.646,-175.823,8.098,148.367
C04534=1212.885,392.241,-79.607,-175.824,8.095,148.367
C04535=1212.888,391.994,-79.572,-175.824,8.092,148.366
C04536=1212.893,391.746,-79.538,-175.825,8.090,148.366
C04537=1212.898,391.499,-79.503,-175.826,8.087,148.365
C04538=1212.901,391.251,-79.469,-175.826,8.085,148.365
C04539=1212.905,391.004,-79.435,-175.827,8.081,148.364
C04540=1212.909,390.755,-79.401,-175.828,8.079,148.364
C04541=1212.913,390.508,-79.367,-175.829,8.076,148.363
C04542=1212.917,390.261,-79.333,-175.830,8.074,148.363
C04543=1212.921,390.013,-79.298,-175.830,8.071,148.363
C04544=1212.926,389.765,-79.264,-175.831,8.068,148.362
C04545=1212.930,389.518,-79.230,-175.832,8.065,148.362
C04546=1212.934,389.270,-79.195,-175.833,8.063,148.361
C04547=1212.937,389.023,-79.161,-175.834,8.061,148.361
C04548=1212.942,388.775,-79.126,-175.834,8.057,148.360
C04549=1212.946,388.527,-79.093,-175.835,8.055,148.360
C04550=1212.950,388.279,-79.058,-175.836,8.052,148.359
C04551=1212.953,388.032,-79.024,-175.837,8.050,148.359
C04552=1212.958,387.784,-78.990,-175.837,8.047,148.358
C04553=1212.962,387.537,-78.956,-175.838,8.044,148.358
C04554=1212.966,387.289,-78.921,-175.839,8.041,148.357
C04555=1212.971,387.041,-78.887,-175.840,8.039,148.357
C04556=1212.974,386.794,-78.853,-175.841,8.037,148.357
C04557=1212.978,386.546,-78.819,-175.842,8.033,148.356
C04558=1212.982,386.299,-78.785,-175.843,8.031,148.356
C04559=1212.987,386.051,-78.750,-175.844,8.028,148.355
C04560=1212.990,385.803,-78.717,-175.844,8.026,148.355
C04561=1212.994,385.556,-78.683,-175.846,8.023,148.354
C04562=1212.999,385.308,-78.648,-175.846,8.020,148.354
C04563=1213.002,385.060,-78.614,-175.848,8.017,148.353
C04564=1213.007,384.812,-78.580,-175.848,8.015,148.353
C04565=1213.011,384.565,-78.547,-175.849,8.012,148.352
C04566=1213.015,384.318,-78.512,-175.850,8.009,148.352
C04567=1213.018,384.070,-78.478,-175.851,8.006,148.352
C04568=1213.023,383.822,-78.444,-175.852,8.003,148.351
C04569=1213.027,383.575,-78.410,-175.853,8.001,148.351
C04570=1213.031,383.327,-78.375,-175.854,7.998,148.350
C04571=1213.035,383.079,-78.342,-175.855,7.995,148.350
C04572=1213.040,382.832,-78.308,-175.856,7.992,148.349
C04573=1213.043,382.584,-78.274,-175.857,7.989,148.349
C04574=1213.047,382.336,-78.240,-175.858,7.986,148.348
C04575=1213.052,382.089,-78.206,-175.858,7.984,148.348
C04576=1213.056,381.842,-78.172,-175.860,7.982,148.348
C04577=1213.060,381.593,-78.138,-175.861,7.979,148.347
C04578=1213.064,381.346,-78.104,-175.862,7.976,148.347
C04579=1213.068,381.099,-78.070,-175.863,7.973,148.346
C04580=1213.072,380.851,-78.036,-175.864,7.970,148.346
C04581=1213.076,380.603,-78.002,-175.865,7.967,148.345
C04582=1213.081,380.355,-77.968,-175.866,7.964,148.345
C04583=1213.084,380.108,-77.935,-175.867,7.961,148.344
C04584=1213.088,379.861,-77.901,-175.868,7.958,148.344
C04585=1213.093,379.612,-77.867,-175.869,7.957,148.344
C04586=1213.096,379.365,-77.833,-175.870,7.953,148.343
C04587=1213.100,379.117,-77.800,-175.871,7.951,148.343
C04588=1213.105,378.870,-77.765,-175.872,7.948,148.342
C04589=1213.109,378.621,-77.732,-175.873,7.945,148.342
C04590=1213.112,378.374,-77.698,-175.875,7.942,148.341
C04591=1213.117,378.126,-77.664,-175.876,7.939,148.341
C04592=1213.121,377.879,-77.630,-175.877,7.937,148.341
C04593=1213.125,377.630,-77.597,-175.878,7.933,148.340
C04594=1213.129,377.383,-77.562,-175.879,7.931,148.340
C04595=1213.133,377.135,-77.529,-175.880,7.928,148.339
C04596=1213.137,376.888,-77.495,-175.881,7.925,148.339
C04597=1213.142,376.640,-77.461,-175.882,7.922,148.339
C04598=1213.145,376.392,-77.427,-175.884,7.919,148.338
C04599=1213.149,376.145,-77.394,-175.885,7.917,148.338
C04600=1213.153,375.897,-77.360,-175.886,7.914,148.337
C04601=1213.158,375.649,-77.326,-175.887,7.911,148.337
C04602=1213.161,375.402,-77.292,-175.888,7.908,148.337
C04603=1213.166,375.154,-77.259,-175.890,7.905,148.336
C04604=1213.170,374.906,-77.225,-175.891,7.902,148.336
C04605=1213.174,374.659,-77.191,-175.892,7.899,148.335
C04606=1213.178,374.411,-77.158,-175.893,7.896,148.335
C04607=1213.182,374.164,-77.124,-175.894,7.893,148.334
C04608=1213.186,373.915,-77.090,-175.896,7.890,148.334
C04609=1213.191,373.667,-77.057,-175.897,7.887,148.334
C04610=1213.194,373.420,-77.023,-175.898,7.884,148.333
C04611=1213.199,373.173,-76.990,-175.900,7.882,148.333
C04612=1213.203,372.925,-76.957,-175.901,7.879,148.333
C04613=1213.207,372.677,-76.922,-175.902,7.876,148.332
C04614=1213.211,372.429,-76.889,-175.903,7.873,148.332
C04615=1213.215,372.181,-76.856,-175.905,7.870,148.331
C04616=1213.219,371.934,-76.822,-175.906,7.867,148.331
C04617=1213.223,371.686,-76.789,-175.907,7.864,148.331
C04618=1213.228,371.438,-76.755,-175.909,7.861,148.330
C04619=1213.232,371.191,-76.722,-175.910,7.859,148.330
C04620=1213.236,370.944,-76.688,-175.911,7.856,148.329
C04621=1213.239,370.695,-76.654,-175.913,7.852,148.329
C04622=1213.243,370.447,-76.621,-175.914,7.850,148.329
C04623=1213.248,370.200,-76.588,-175.916,7.847,148.328
C04624=1213.251,369.953,-76.554,-175.917,7.844,148.328
C04625=1213.256,369.705,-76.520,-175.918,7.841,148.328
C04626=1213.260,369.457,-76.487,-175.919,7.838,148.327
C04627=1213.265,369.209,-76.454,-175.921,7.835,148.327
C04628=1213.269,368.961,-76.421,-175.923,7.832,148.327
C04629=1213.272,368.714,-76.387,-175.924,7.829,148.326
C04630=1213.276,368.466,-76.354,-175.925,7.827,148.326
C04631=1213.280,368.218,-76.320,-175.927,7.823,148.325
C04632=1213.284,367.970,-76.287,-175.928,7.820,148.325
C04633=1213.288,367.723,-76.254,-175.930,7.818,148.325
C04634=1213.293,367.475,-76.220,-175.931,7.815,148.324
C04635=1213.298,367.195,-76.183,-175.932,7.811,148.324
C04636=1213.302,366.915,-76.145,-175.934,7.807,148.323
C04637=1213.307,366.635,-76.107,-175.936,7.805,148.323
C04638=1213.312,366.354,-76.070,-175.938,7.801,148.323
C04639=1213.316,366.106,-76.036,-175.939,7.798,148.322
C04640=1213.320,365.858,-76.003,-175.941,7.795,148.322
C04641=1213.324,365.611,-75.970,-175.942,7.792,148.322
C04642=1213.328,365.363,-75.937,-175.943,7.789,148.321
C04643=1213.332,365.115,-75.904,-175.945,7.787,148.321
C04644=1213.336,364.868,-75.871,-175.947,7.783,148.321
C04645=1213.340,364.620,-75.837,-175.948,7.780,148.320
C04646=1213.344,364.373,-75.804,-175.950,7.778,148.320
C04647=1213.349,364.124,-75.771,-175.951,7.774,148.320
C04648=1213.353,363.877,-75.738,-175.953,7.772,148.319
C04649=1213.357,363.629,-75.705,-175.954,7.769,148.319
C04650=1213.361,363.381,-75.672,-175.956,7.765,148.319
C04651=1213.365,363.133,-75.639,-175.958,7.763,148.319
C04652=1213.370,362.886,-75.605,-175.959,7.760,148.318
C04653=1213.374,362.638,-75.572,-175.961,7.757,148.318
C04654=1213.377,362.391,-75.540,-175.962,7.754,148.318
C04655=1213.381,362.143,-75.507,-175.964,7.751,148.317
C04656=1213.385,361.895,-75.473,-175.966,7.748,148.317
C04657=1213.390,361.647,-75.440,-175.967,7.745,148.317
C04658=1213.394,361.400,-75.407,-175.968,7.742,148.316
C04659=1213.398,361.152,-75.374,-175.971,7.739,148.316
C04660=1213.402,360.904,-75.341,-175.972,7.736,148.316
C04661=1213.406,360.656,-75.308,-175.973,7.734,148.316
C04662=1213.410,360.408,-75.275,-175.975,7.730,148.315
C04663=1213.415,360.160,-75.242,-175.977,7.727,148.315
C04664=1213.419,359.913,-75.209,-175.979,7.724,148.314
C04665=1213.422,359.665,-75.176,-175.980,7.721,148.314
C04666=1213.427,359.417,-75.144,-175.981,7.719,148.314
C04667=1213.431,359.169,-75.111,-175.984,7.715,148.314
C04668=1213.435,358.921,-75.078,-175.985,7.713,148.313
C04669=1213.439,358.674,-75.044,-175.986,7.710,148.313
C04670=1213.443,358.425,-75.012,-175.989,7.706,148.313
C04671=1213.448,358.178,-74.979,-175.990,7.704,148.313
C04672=1213.451,357.930,-74.946,-175.992,7.700,148.312
C04673=1213.455,357.682,-74.913,-175.994,7.698,148.312
C04674=1213.460,357.434,-74.881,-175.995,7.695,148.312
C04675=1213.464,357.186,-74.847,-175.997,7.692,148.311
C04676=1213.468,356.939,-74.814,-175.999,7.689,148.311
C04677=1213.472,356.691,-74.782,-176.001,7.686,148.311
C04678=1213.476,356.443,-74.749,-176.002,7.683,148.311
C04679=1213.480,356.196,-74.717,-176.004,7.680,148.310
C04680=1213.485,355.947,-74.684,-176.006,7.677,148.310
C04681=1213.488,355.700,-74.652,-176.007,7.674,148.310
C04682=1213.492,355.452,-74.618,-176.009,7.671,148.310
C04683=1213.497,355.204,-74.586,-176.011,7.668,148.309
C04684=1213.501,354.956,-74.553,-176.013,7.665,148.309
C04685=1213.505,354.708,-74.521,-176.014,7.662,148.309
C04686=1213.509,354.460,-74.488,-176.016,7.660,148.309
C04687=1213.513,354.213,-74.455,-176.018,7.656,148.308
C04688=1213.518,353.965,-74.423,-176.020,7.654,148.308
C04689=1213.521,353.718,-74.390,-176.022,7.650,148.308
C04690=1213.526,353.469,-74.358,-176.023,7.648,148.308
C04691=1213.530,353.222,-74.324,-176.026,7.644,148.307
C04692=1213.534,352.974,-74.293,-176.027,7.642,148.307
C04693=1213.538,352.726,-74.259,-176.029,7.639,148.307
C04694=1213.542,352.477,-74.227,-176.031,7.636,148.307
C04695=1213.547,352.230,-74.194,-176.032,7.633,148.306
C04696=1213.551,351.982,-74.162,-176.034,7.630,148.306
C04697=1213.555,351.735,-74.129,-176.036,7.627,148.306
C04698=1213.559,351.486,-74.097,-176.038,7.624,148.306
C04699=1213.563,351.239,-74.064,-176.040,7.621,148.306
C04700=1213.567,350.991,-74.032,-176.042,7.618,148.305
C04701=1213.571,350.743,-74.000,-176.044,7.615,148.305
C04702=1213.576,350.496,-73.967,-176.045,7.612,148.305
C04703=1213.580,350.247,-73.935,-176.047,7.609,148.305
C04704=1213.583,350.000,-73.902,-176.049,7.607,148.304
C04705=1213.588,349.751,-73.870,-176.051,7.603,148.304
C04706=1213.593,349.504,-73.838,-176.053,7.601,148.304
C04707=1213.596,349.256,-73.805,-176.055,7.598,148.304
C04708=1213.601,349.008,-73.773,-176.056,7.595,148.304
C04709=1213.605,348.760,-73.741,-176.059,7.592,148.303
C04710=1213.609,348.512,-73.708,-176.060,7.589,148.303
C04711=1213.613,348.265,-73.676,-176.063,7.586,148.303
C04712=1213.617,348.017,-73.644,-176.064,7.583,148.303
C04713=1213.622,347.769,-73.610,-176.066,7.580,148.302
C04714=1213.625,347.521,-73.579,-176.068,7.577,148.302
C04715=1213.630,347.273,-73.547,-176.070,7.574,148.302
C04716=1213.634,347.025,-73.515,-176.072,7.572,148.302
C04717=1213.638,346.777,-73.482,-176.074,7.569,148.302
C04718=1213.642,346.529,-73.450,-176.076,7.566,148.301
C04719=1213.647,346.282,-73.418,-176.077,7.563,148.301
C04720=1213.651,346.034,-73.386,-176.080,7.560,148.301
C04721=1213.655,345.785,-73.353,-176.081,7.557,148.301
C04722=1213.658,345.538,-73.321,-176.083,7.554,148.301
C04723=1213.663,345.290,-73.289,-176.085,7.551,148.301
C04724=1213.667,345.042,-73.257,-176.087,7.548,148.300
C04725=1213.672,344.794,-73.224,-176.089,7.546,148.300
C04726=1213.676,344.546,-73.193,-176.091,7.542,148.300
C04727=1213.680,344.298,-73.161,-176.093,7.540,148.300
C04728=1213.684,344.050,-73.129,-176.095,7.537,148.300
C04729=1213.688,343.802,-73.097,-176.097,7.534,148.300
C04730=1213.693,343.555,-73.064,-176.099,7.531,148.299
C04731=1213.696,343.307,-73.032,-176.101,7.528,148.299
C04732=1213.701,343.059,-73.000,-176.103,7.525,148.299
C04733=1213.705,342.811,-72.968,-176.105,7.522,148.299
C04734=1213.709,342.563,-72.936,-176.107,7.519,148.298
C04735=1213.713,342.315,-72.904,-176.109,7.517,148.298
C04736=1213.717,342.068,-72.872,-176.111,7.514,148.298
C04737=1213.722,341.819,-72.840,-176.113,7.511,148.298
C04738=1213.726,341.571,-72.808,-176.115,7.508,148.298
C04739=1213.731,341.293,-72.772,-176.117,7.504,148.298
C04740=1213.735,341.015,-72.737,-176.119,7.502,148.297
C04741=1213.740,340.737,-72.701,-176.122,7.499,148.297
C04742=1213.745,340.460,-72.665,-176.124,7.495,148.297
C04743=1213.749,340.211,-72.633,-176.126,7.492,148.297
C04744=1213.753,339.963,-72.601,-176.128,7.490,148.297
C04745=1213.757,339.715,-72.570,-176.130,7.486,148.297
C04746=1213.761,339.467,-72.538,-176.132,7.484,148.297
C04747=1213.766,339.219,-72.506,-176.134,7.481,148.296
C04748=1213.770,338.972,-72.474,-176.136,7.478,148.296
C04749=1213.774,338.724,-72.443,-176.138,7.475,148.296
C04750=1213.779,338.476,-72.411,-176.140,7.473,148.296
C04751=1213.782,338.228,-72.379,-176.142,7.469,148.296
C04752=1213.786,337.980,-72.347,-176.144,7.467,148.296
C04753=1213.791,337.732,-72.316,-176.146,7.463,148.295
C04754=1213.795,337.484,-72.284,-176.148,7.461,148.295
C04755=1213.799,337.236,-72.252,-176.151,7.458,148.295
C04756=1213.803,336.988,-72.220,-176.152,7.455,148.295
C04757=1213.807,336.740,-72.189,-176.155,7.452,148.295
C04758=1213.812,336.492,-72.157,-176.156,7.450,148.295
C04759=1213.816,336.244,-72.125,-176.159,7.446,148.295
C04760=1213.820,335.997,-72.094,-176.161,7.444,148.295
C04761=1213.824,335.749,-72.062,-176.163,7.441,148.294
C04762=1213.829,335.501,-72.031,-176.165,7.438,148.294
C04763=1213.833,335.252,-71.999,-176.167,7.435,148.294
C04764=1213.837,335.004,-71.967,-176.169,7.433,148.294
C04765=1213.841,334.756,-71.936,-176.171,7.429,148.294
C04766=1213.845,334.508,-71.904,-176.173,7.427,148.294
C04767=1213.849,334.261,-71.873,-176.175,7.424,148.294
C04768=1213.853,334.012,-71.842,-176.177,7.421,148.294
C04769=1213.858,333.765,-71.810,-176.180,7.418,148.294
C04770=1213.862,333.517,-71.778,-176.181,7.416,148.293
C04771=1213.867,333.269,-71.747,-176.184,7.413,148.293
C04772=1213.870,333.021,-71.715,-176.186,7.409,148.293
C04773=1213.875,332.773,-71.684,-176.188,7.407,148.293
C04774=1213.879,332.525,-71.653,-176.191,7.404,148.293
C04775=1213.883,332.277,-71.621,-176.192,7.401,148.293
C04776=1213.887,332.029,-71.590,-176.195,7.398,148.293
C04777=1213.891,331.781,-71.558,-176.197,7.396,148.293
C04778=1213.895,331.533,-71.527,-176.199,7.393,148.293
C04779=1213.900,331.285,-71.496,-176.201,7.390,148.292
C04780=1213.904,331.036,-71.464,-176.203,7.387,148.292
C04781=1213.909,330.789,-71.433,-176.205,7.385,148.292
C04782=1213.913,330.540,-71.402,-176.207,7.381,148.292
C04783=1213.917,330.293,-71.370,-176.210,7.379,148.292
C04784=1213.921,330.044,-71.339,-176.212,7.376,148.292
C04785=1213.925,329.797,-71.307,-176.214,7.373,148.292
C04786=1213.929,329.548,-71.276,-176.216,7.370,148.292
C04787=1213.934,329.301,-71.245,-176.218,7.368,148.292
C04788=1213.938,329.053,-71.214,-176.220,7.364,148.291
C04789=1213.942,328.804,-71.183,-176.222,7.362,148.292
C04790=1213.947,328.557,-71.151,-176.225,7.359,148.291
C04791=1213.951,328.308,-71.120,-176.227,7.357,148.291
C04792=1213.955,328.061,-71.089,-176.229,7.353,148.291
C04793=1213.959,327.812,-71.058,-176.231,7.351,148.291
C04794=1213.964,327.564,-71.027,-176.233,7.348,148.291
C04795=1213.968,327.317,-70.995,-176.235,7.346,148.291
C04796=1213.971,327.069,-70.965,-176.238,7.343,148.291
C04797=1213.976,326.821,-70.934,-176.240,7.340,148.291
C04798=1213.979,326.573,-70.902,-176.242,7.337,148.291
C04799=1213.984,326.325,-70.872,-176.244,7.334,148.291
C04800=1213.989,326.077,-70.841,-176.247,7.331,148.291
C04801=1213.993,325.828,-70.810,-176.248,7.329,148.290
C04802=1213.997,325.581,-70.778,-176.251,7.326,148.290
C04803=1214.001,325.332,-70.747,-176.254,7.323,148.290
C04804=1214.006,325.084,-70.716,-176.255,7.320,148.290
C04805=1214.009,324.836,-70.686,-176.258,7.317,148.290
C04806=1214.013,324.588,-70.654,-176.260,7.315,148.290
C04807=1214.018,324.340,-70.624,-176.262,7.312,148.290
C04808=1214.022,324.093,-70.593,-176.264,7.309,148.290
C04809=1214.026,323.844,-70.562,-176.267,7.306,148.290
C04810=1214.031,323.596,-70.531,-176.269,7.304,148.290
C04811=1214.035,323.349,-70.500,-176.271,7.301,148.290
C04812=1214.039,323.100,-70.469,-176.273,7.298,148.290
C04813=1214.043,322.852,-70.438,-176.276,7.295,148.290
C04814=1214.047,322.604,-70.407,-176.277,7.293,148.290
C04815=1214.052,322.356,-70.376,-176.280,7.290,148.290
C04816=1214.056,322.108,-70.346,-176.282,7.288,148.290
C04817=1214.060,321.860,-70.315,-176.284,7.284,148.289
C04818=1214.064,321.611,-70.284,-176.286,7.282,148.290
C04819=1214.069,321.363,-70.253,-176.289,7.279,148.290
C04820=1214.074,321.115,-70.223,-176.291,7.276,148.289
C04821=1214.077,320.867,-70.192,-176.293,7.273,148.289
C04822=1214.081,320.619,-70.161,-176.296,7.271,148.289
C04823=1214.086,320.371,-70.131,-176.298,7.268,148.289
C04824=1214.089,320.123,-70.100,-176.300,7.266,148.289
C04825=1214.094,319.875,-70.069,-176.303,7.263,148.289
C04826=1214.099,319.627,-70.038,-176.305,7.260,148.289
C04827=1214.103,319.379,-70.008,-176.307,7.257,148.289
C04828=1214.106,319.131,-69.977,-176.309,7.255,148.289
C04829=1214.111,318.883,-69.946,-176.312,7.252,148.289
C04830=1214.116,318.635,-69.916,-176.314,7.250,148.289
C04831=1214.120,318.387,-69.885,-176.316,7.246,148.289
C04832=1214.124,318.138,-69.854,-176.318,7.244,148.289
C04833=1214.128,317.890,-69.824,-176.321,7.241,148.289
C04834=1214.132,317.643,-69.793,-176.323,7.239,148.289
C04835=1214.137,317.395,-69.763,-176.325,7.235,148.289
C04836=1214.141,317.146,-69.732,-176.327,7.233,148.289
C04837=1214.145,316.898,-69.702,-176.330,7.230,148.289
C04838=1214.150,316.650,-69.671,-176.333,7.227,148.289
C04839=1214.153,316.402,-69.641,-176.334,7.225,148.289
C04840=1214.157,316.154,-69.610,-176.337,7.222,148.289
C04841=1214.162,315.906,-69.579,-176.339,7.219,148.289
C04842=1214.166,315.657,-69.550,-176.342,7.216,148.289
C04843=1214.171,315.382,-69.516,-176.344,7.214,148.289
C04844=1214.176,315.106,-69.481,-176.346,7.211,148.289
C04845=1214.180,314.830,-69.448,-176.349,7.208,148.289
C04846=1214.185,314.554,-69.414,-176.351,7.205,148.289
C04847=1214.190,314.305,-69.384,-176.354,7.202,148.289
C04848=1214.194,314.058,-69.354,-176.356,7.199,148.289
C04849=1214.198,313.810,-69.323,-176.359,7.196,148.289
C04850=1214.202,313.561,-69.293,-176.361,7.194,148.289
C04851=1214.206,313.313,-69.262,-176.364,7.191,148.289
C04852=1214.210,313.065,-69.232,-176.365,7.189,148.289
C04853=1214.215,312.817,-69.202,-176.368,7.186,148.289
C04854=1214.219,312.569,-69.172,-176.370,7.183,148.289
C04855=1214.224,312.321,-69.141,-176.373,7.180,148.289
C04856=1214.227,312.072,-69.111,-176.375,7.178,148.289
C04857=1214.232,311.824,-69.081,-176.377,7.175,148.289
C04858=1214.236,311.576,-69.051,-176.380,7.173,148.289
C04859=1214.241,311.328,-69.020,-176.382,7.169,148.289
C04860=1214.245,311.080,-68.990,-176.384,7.167,148.289
C04861=1214.250,310.832,-68.960,-176.387,7.164,148.289
C04862=1214.253,310.584,-68.930,-176.389,7.162,148.289
C04863=1214.258,310.336,-68.901,-176.391,7.159,148.289
C04864=1214.262,310.088,-68.870,-176.393,7.157,148.289
C04865=1214.266,309.839,-68.840,-176.396,7.154,148.289
C04866=1214.270,309.591,-68.809,-176.398,7.152,148.289
C04867=1214.275,309.343,-68.780,-176.401,7.148,148.289
C04868=1214.279,309.095,-68.749,-176.403,7.146,148.289
C04869=1214.283,308.846,-68.720,-176.406,7.143,148.289
C04870=1214.287,308.599,-68.689,-176.407,7.141,148.289
C04871=1214.292,308.350,-68.659,-176.410,7.138,148.289
C04872=1214.296,308.102,-68.630,-176.412,7.135,148.289
C04873=1214.300,307.854,-68.600,-176.415,7.132,148.289
C04874=1214.305,307.606,-68.570,-176.417,7.130,148.289
C04875=1214.309,307.358,-68.540,-176.419,7.128,148.289
C04876=1214.313,307.110,-68.510,-176.422,7.125,148.289
C04877=1214.318,306.861,-68.480,-176.424,7.123,148.289
C04878=1214.322,306.613,-68.450,-176.427,7.120,148.289
C04879=1214.326,306.365,-68.420,-176.429,7.118,148.289
C04880=1214.331,306.117,-68.390,-176.431,7.114,148.289
C04881=1214.335,305.869,-68.360,-176.433,7.112,148.289
C04882=1214.339,305.621,-68.331,-176.436,7.109,148.289
C04883=1214.343,305.372,-68.301,-176.438,7.107,148.289
C04884=1214.348,305.125,-68.271,-176.441,7.104,148.289
C04885=1214.352,304.876,-68.241,-176.443,7.102,148.289
C04886=1214.356,304.628,-68.212,-176.446,7.099,148.289
C04887=1214.361,304.379,-68.182,-176.448,7.097,148.289
C04888=1214.365,304.132,-68.151,-176.450,7.094,148.289
C04889=1214.369,303.883,-68.122,-176.453,7.091,148.289
C04890=1214.373,303.635,-68.093,-176.455,7.088,148.289
C04891=1214.378,303.387,-68.063,-176.457,7.086,148.289
C04892=1214.383,303.138,-68.033,-176.460,7.083,148.289
C04893=1214.386,302.891,-68.003,-176.462,7.081,148.289
C04894=1214.391,302.642,-67.973,-176.465,7.078,148.289
C04895=1214.395,302.394,-67.944,-176.467,7.076,148.290
C04896=1214.399,302.146,-67.915,-176.469,7.073,148.290
C04897=1214.404,301.897,-67.884,-176.472,7.070,148.290
C04898=1214.408,301.649,-67.855,-176.474,7.068,148.290
C04899=1214.412,301.401,-67.826,-176.477,7.065,148.290
C04900=1214.416,301.153,-67.796,-176.479,7.063,148.290
C04901=1214.421,300.904,-67.767,-176.481,7.060,148.290
C04902=1214.425,300.657,-67.736,-176.484,7.058,148.290
C04903=1214.429,300.408,-67.707,-176.487,7.055,148.290
C04904=1214.434,300.160,-67.677,-176.489,7.053,148.290
C04905=1214.438,299.912,-67.648,-176.491,7.050,148.290
C04906=1214.443,299.664,-67.618,-176.494,7.047,148.290
C04907=1214.447,299.416,-67.589,-176.496,7.044,148.290
C04908=1214.451,299.167,-67.560,-176.498,7.042,148.290
C04909=1214.455,298.919,-67.530,-176.500,7.040,148.290
C04910=1214.459,298.671,-67.501,-176.503,7.037,148.290
C04911=1214.463,298.423,-67.471,-176.505,7.035,148.290
C04912=1214.468,298.174,-67.442,-176.508,7.032,148.290
C04913=1214.473,297.926,-67.413,-176.510,7.030,148.290
C04914=1214.477,297.678,-67.384,-176.513,7.027,148.291
C04915=1214.481,297.430,-67.354,-176.515,7.025,148.291
C04916=1214.485,297.181,-67.325,-176.518,7.022,148.291
C04917=1214.489,296.933,-67.296,-176.520,7.019,148.291
C04918=1214.494,296.685,-67.266,-176.522,7.017,148.291
C04919=1214.498,296.437,-67.237,-176.525,7.014,148.291
C04920=1214.503,296.189,-67.208,-176.527,7.012,148.291
C04921=1214.507,295.941,-67.178,-176.530,7.009,148.291
C04922=1214.511,295.692,-67.149,-176.532,7.007,148.291
C04923=1214.515,295.444,-67.120,-176.535,7.004,148.291
C04924=1214.520,295.195,-67.090,-176.537,7.002,148.291
C04925=1214.524,294.947,-67.061,-176.539,7.000,148.291
C04926=1214.529,294.699,-67.032,-176.542,6.997,148.291
C04927=1214.533,294.451,-67.003,-176.544,6.994,148.291
C04928=1214.537,294.202,-66.974,-176.547,6.991,148.291
C04929=1214.541,293.954,-66.944,-176.549,6.989,148.292
C04930=1214.546,293.706,-66.915,-176.552,6.986,148.292
C04931=1214.550,293.458,-66.887,-176.554,6.984,148.292
C04932=1214.554,293.210,-66.858,-176.556,6.982,148.292
C04933=1214.558,292.961,-66.828,-176.559,6.979,148.292
C04934=1214.563,292.712,-66.799,-176.562,6.977,148.292
C04935=1214.567,292.464,-66.770,-176.564,6.974,148.292
C04936=1214.572,292.217,-66.741,-176.566,6.972,148.292
C04937=1214.576,291.968,-66.712,-176.569,6.969,148.292
C04938=1214.580,291.719,-66.683,-176.571,6.967,148.292
C04939=1214.584,291.472,-66.654,-176.574,6.965,148.293
C04940=1214.589,291.223,-66.625,-176.576,6.962,148.293
C04941=1214.593,290.975,-66.596,-176.579,6.959,148.293
C04942=1214.598,290.726,-66.567,-176.581,6.956,148.293
C04943=1214.602,290.478,-66.538,-176.583,6.954,148.293
C04944=1214.606,290.231,-66.509,-176.586,6.952,148.293
C04945=1214.610,289.982,-66.481,-176.589,6.949,148.293
C04946=1214.615,289.733,-66.451,-176.591,6.947,148.293
C04947=1214.619,289.459,-66.419,-176.593,6.944,148.293
C04948=1214.624,289.185,-66.388,-176.597,6.941,148.293
C04949=1214.629,288.910,-66.356,-176.599,6.938,148.293
C04950=1214.634,288.637,-66.324,-176.601,6.936,148.294
C04951=1214.639,288.389,-66.295,-176.605,6.933,148.294
C04952=1214.643,288.140,-66.266,-176.607,6.931,148.294
C04953=1214.647,287.891,-66.237,-176.609,6.928,148.294
C04954=1214.651,287.644,-66.209,-176.611,6.926,148.294
C04955=1214.656,287.395,-66.180,-176.614,6.924,148.294
C04956=1214.660,287.146,-66.151,-176.617,6.921,148.294
C04957=1214.664,286.899,-66.123,-176.619,6.919,148.294
C04958=1214.669,286.650,-66.094,-176.621,6.917,148.294
C04959=1214.673,286.402,-66.065,-176.624,6.914,148.295
C04960=1214.677,286.154,-66.037,-176.626,6.912,148.295
C04961=1214.682,285.905,-66.008,-176.629,6.909,148.295
C04962=1214.686,285.657,-65.979,-176.632,6.907,148.295
C04963=1214.690,285.409,-65.951,-176.634,6.905,148.295
C04964=1214.695,285.160,-65.922,-176.636,6.902,148.295
C04965=1214.699,284.912,-65.893,-176.638,6.899,148.295
C04966=1214.703,284.664,-65.865,-176.642,6.897,148.295
C04967=1214.708,284.415,-65.836,-176.644,6.894,148.295
C04968=1214.713,284.168,-65.807,-176.646,6.892,148.296
C04969=1214.716,283.919,-65.779,-176.649,6.890,148.296
C04970=1214.721,283.670,-65.750,-176.651,6.887,148.296
C04971=1214.725,283.422,-65.722,-176.653,6.885,148.296
C04972=1214.730,283.173,-65.694,-176.656,6.882,148.296
C04973=1214.735,282.926,-65.665,-176.659,6.880,148.296
C04974=1214.738,282.677,-65.636,-176.661,6.877,148.296
C04975=1214.743,282.428,-65.608,-176.663,6.875,148.296
C04976=1214.747,282.180,-65.580,-176.666,6.873,148.297
C04977=1214.752,281.931,-65.551,-176.669,6.870,148.297
C04978=1214.756,281.684,-65.523,-176.671,6.868,148.297
C04979=1214.760,281.435,-65.494,-176.673,6.866,148.297
C04980=1214.764,281.187,-65.466,-176.676,6.863,148.297
C04981=1214.769,280.939,-65.437,-176.678,6.861,148.297
C04982=1214.773,280.690,-65.409,-176.681,6.859,148.297
C04983=1214.778,280.442,-65.381,-176.684,6.856,148.297
C04984=1214.782,280.193,-65.353,-176.686,6.854,148.297
C04985=1214.787,279.945,-65.324,-176.688,6.852,148.298
C04986=1214.790,279.696,-65.296,-176.691,6.849,148.298
C04987=1214.795,279.449,-65.267,-176.694,6.847,148.298
C04988=1214.799,279.200,-65.239,-176.696,6.845,148.298
C04989=1214.804,278.952,-65.211,-176.698,6.842,148.298
C04990=1214.808,278.704,-65.183,-176.701,6.840,148.298
C04991=1214.813,278.455,-65.154,-176.704,6.837,148.298
C04992=1214.817,278.207,-65.126,-176.706,6.834,148.299
C04993=1214.821,277.959,-65.098,-176.708,6.833,148.299
C04994=1214.825,277.710,-65.069,-176.711,6.830,148.299
C04995=1214.830,277.462,-65.042,-176.713,6.827,148.299
C04996=1214.835,277.213,-65.014,-176.716,6.826,148.299
C04997=1214.839,276.965,-64.986,-176.718,6.822,148.299
C04998=1214.843,276.716,-64.958,-176.721,6.821,148.300
C04999=1214.848,276.468,-64.929,-176.723,6.818,148.300
C05000=1214.852,276.219,-64.901,-176.726,6.815,148.300
C05001=1214.856,275.972,-64.873,-176.728,6.813,148.300
C05002=1214.860,275.723,-64.845,-176.731,6.811,148.300
C05003=1214.865,275.475,-64.817,-176.733,6.809,148.300
C05004=1214.868,275.226,-64.789,-176.736,6.806,148.300
C05005=1214.874,274.977,-64.761,-176.738,6.804,148.300
C05006=1214.878,274.730,-64.733,-176.741,6.802,148.301
C05007=1214.882,274.481,-64.705,-176.743,6.799,148.301
C05008=1214.887,274.233,-64.677,-176.746,6.797,148.301
C05009=1214.891,273.984,-64.649,-176.748,6.795,148.301
C05010=1214.895,273.736,-64.621,-176.751,6.792,148.301
C05011=1214.900,273.487,-64.593,-176.753,6.790,148.301
C05012=1214.904,273.239,-64.565,-176.755,6.788,148.302
C05013=1214.909,272.991,-64.537,-176.759,6.785,148.302
C05014=1214.912,272.743,-64.509,-176.761,6.783,148.302
C05015=1214.918,272.494,-64.482,-176.763,6.781,148.302
C05016=1214.922,272.245,-64.453,-176.766,6.778,148.302
C05017=1214.926,271.997,-64.426,-176.768,6.776,148.302
C05018=1214.931,271.749,-64.399,-176.771,6.774,148.303
C05019=1214.935,271.500,-64.370,-176.773,6.772,148.303
C05020=1214.939,271.252,-64.342,-176.776,6.769,148.303
C05021=1214.944,271.003,-64.315,-176.778,6.767,148.303
C05022=1214.948,270.755,-64.287,-176.781,6.765,148.303
C05023=1214.952,270.507,-64.259,-176.784,6.762,148.303
C05024=1214.957,270.258,-64.231,-176.786,6.760,148.304
C05025=1214.961,270.010,-64.203,-176.788,6.758,148.304
C05026=1214.966,269.761,-64.176,-176.791,6.756,148.304
C05027=1214.970,269.513,-64.148,-176.794,6.753,148.304
C05028=1214.974,269.265,-64.120,-176.796,6.751,148.304
C05029=1214.979,269.016,-64.093,-176.798,6.749,148.304
C05030=1214.983,268.767,-64.065,-176.801,6.746,148.304
C05031=1214.988,268.519,-64.037,-176.804,6.744,148.305
C05032=1214.992,268.271,-64.010,-176.806,6.742,148.305
C05033=1214.996,268.022,-63.982,-176.808,6.740,148.305
C05034=1215.001,267.774,-63.954,-176.811,6.737,148.305
C05035=1215.005,267.525,-63.927,-176.814,6.735,148.305
C05036=1215.010,267.278,-63.900,-176.816,6.733,148.306
C05037=1215.014,267.028,-63.872,-176.818,6.731,148.306
C05038=1215.018,266.780,-63.844,-176.821,6.728,148.306
C05039=1215.023,266.532,-63.817,-176.824,6.726,148.306
C05040=1215.027,266.283,-63.789,-176.826,6.724,148.306
C05041=1215.032,266.035,-63.762,-176.829,6.721,148.306
C05042=1215.036,265.786,-63.735,-176.831,6.719,148.307
C05043=1215.041,265.538,-63.707,-176.834,6.717,148.307
C05044=1215.045,265.289,-63.679,-176.836,6.715,148.307
C05045=1215.049,265.041,-63.652,-176.839,6.712,148.307
C05046=1215.054,264.793,-63.624,-176.841,6.710,148.307
C05047=1215.059,264.544,-63.597,-176.844,6.708,148.308
C05048=1215.062,264.296,-63.569,-176.846,6.706,148.308
C05049=1215.067,264.047,-63.542,-176.849,6.703,148.308
C05050=1215.072,263.799,-63.515,-176.851,6.701,148.308
C05051=1215.076,263.526,-63.485,-176.854,6.699,148.308
C05052=1215.081,263.254,-63.455,-176.857,6.697,148.309
C05053=1215.085,262.981,-63.425,-176.859,6.694,148.309
C05054=1215.091,262.708,-63.395,-176.862,6.692,148.309
C05055=1215.095,262.459,-63.368,-176.865,6.690,148.309
C05056=1215.100,262.211,-63.341,-176.868,6.687,148.309
C05057=1215.105,261.963,-63.314,-176.870,6.685,148.310
C05058=1215.108,261.714,-63.285,-176.872,6.683,148.310
C05059=1215.113,261.465,-63.258,-176.875,6.681,148.310
C05060=1215.117,261.217,-63.232,-176.877,6.679,148.310
C05061=1215.122,260.969,-63.205,-176.880,6.676,148.310
C05062=1215.126,260.720,-63.178,-176.882,6.674,148.310
C05063=1215.130,260.472,-63.150,-176.885,6.672,148.311
C05064=1215.135,260.223,-63.123,-176.887,6.670,148.311
C05065=1215.139,259.975,-63.095,-176.890,6.667,148.311
C05066=1215.144,259.726,-63.068,-176.893,6.665,148.311
C05067=1215.149,259.478,-63.041,-176.895,6.663,148.311
C05068=1215.152,259.230,-63.015,-176.898,6.661,148.312
C05069=1215.157,258.980,-62.987,-176.900,6.659,148.312
C05070=1215.161,258.732,-62.960,-176.903,6.656,148.312
C05071=1215.166,258.483,-62.933,-176.905,6.654,148.312
C05072=1215.170,258.235,-62.906,-176.908,6.652,148.312
C05073=1215.175,257.987,-62.878,-176.910,6.650,148.313
C05074=1215.179,257.739,-62.852,-176.912,6.648,148.313
C05075=1215.183,257.490,-62.825,-176.916,6.645,148.313
C05076=1215.188,257.242,-62.798,-176.918,6.643,148.313
C05077=1215.192,256.993,-62.770,-176.920,6.641,148.313
C05078=1215.196,256.744,-62.744,-176.922,6.639,148.314
C05079=1215.201,256.496,-62.717,-176.925,6.637,148.314
C05080=1215.205,256.247,-62.690,-176.928,6.635,148.314
C05081=1215.210,255.999,-62.663,-176.930,6.632,148.314
C05082=1215.215,255.750,-62.636,-176.933,6.631,148.315
C05083=1215.219,255.502,-62.610,-176.935,6.628,148.315
C05084=1215.224,255.253,-62.583,-176.938,6.627,148.315
C05085=1215.228,255.005,-62.556,-176.941,6.624,148.315
C05086=1215.232,254.756,-62.529,-176.943,6.622,148.315
C05087=1215.237,254.508,-62.502,-176.946,6.620,148.316
C05088=1215.241,254.259,-62.475,-176.948,6.618,148.316
C05089=1215.245,254.011,-62.448,-176.950,6.616,148.316
C05090=1215.249,253.762,-62.421,-176.954,6.613,148.316
C05091=1215.254,253.513,-62.395,-176.956,6.611,148.316
C05092=1215.258,253.265,-62.369,-176.958,6.609,148.317
C05093=1215.263,253.016,-62.342,-176.961,6.607,148.317
C05094=1215.268,252.768,-62.314,-176.963,6.605,148.317
C05095=1215.272,252.520,-62.288,-176.966,6.603,148.317
C05096=1215.276,252.271,-62.261,-176.968,6.600,148.317
C05097=1215.281,252.022,-62.235,-176.971,6.598,148.318
C05098=1215.285,251.774,-62.208,-176.974,6.596,148.318
C05099=1215.290,251.525,-62.181,-176.976,6.594,148.318
C05100=1215.294,251.277,-62.154,-176.978,6.592,148.318
C05101=1215.299,251.028,-62.128,-176.981,6.590,148.319
C05102=1215.303,250.779,-62.101,-176.984,6.587,148.319
C05103=1215.307,250.531,-62.075,-176.986,6.585,148.319
C05104=1215.312,250.282,-62.048,-176.989,6.583,148.319
C05105=1215.316,250.034,-62.022,-176.991,6.581,148.319
C05106=1215.321,249.786,-61.995,-176.994,6.580,148.320
C05107=1215.326,249.536,-61.969,-176.996,6.577,148.320
C05108=1215.330,249.288,-61.942,-176.999,6.575,148.320
C05109=1215.334,249.040,-61.915,-177.002,6.573,148.320
C05110=1215.339,248.791,-61.889,-177.004,6.571,148.321
C05111=1215.343,248.542,-61.862,-177.006,6.569,148.321
C05112=1215.347,248.294,-61.836,-177.009,6.567,148.321
C05113=1215.353,248.046,-61.810,-177.011,6.565,148.321
C05114=1215.357,247.798,-61.783,-177.014,6.563,148.322
C05115=1215.362,247.549,-61.757,-177.017,6.560,148.322
C05116=1215.365,247.300,-61.730,-177.019,6.558,148.322
C05117=1215.370,247.051,-61.704,-177.022,6.556,148.322
C05118=1215.374,246.803,-61.678,-177.024,6.554,148.323
C05119=1215.379,246.554,-61.651,-177.027,6.552,148.323
C05120=1215.383,246.306,-61.625,-177.029,6.550,148.323
C05121=1215.388,246.057,-61.598,-177.032,6.548,148.323
C05122=1215.392,245.808,-61.572,-177.034,6.546,148.323
C05123=1215.396,245.560,-61.546,-177.037,6.543,148.324
C05124=1215.401,245.311,-61.519,-177.040,6.542,148.324
C05125=1215.406,245.063,-61.494,-177.042,6.539,148.324
C05126=1215.410,244.815,-61.467,-177.044,6.537,148.324
C05127=1215.415,244.566,-61.441,-177.047,6.536,148.325
C05128=1215.419,244.318,-61.415,-177.050,6.534,148.325
C05129=1215.424,244.068,-61.388,-177.052,6.532,148.325
C05130=1215.428,243.820,-61.362,-177.054,6.530,148.325
C05131=1215.432,243.571,-61.335,-177.058,6.527,148.326
C05132=1215.437,243.322,-61.310,-177.060,6.525,148.326
C05133=1215.441,243.075,-61.284,-177.062,6.523,148.326
C05134=1215.446,242.826,-61.257,-177.065,6.521,148.326
C05135=1215.450,242.577,-61.231,-177.067,6.519,148.326
C05136=1215.454,242.329,-61.205,-177.070,6.517,148.327
C05137=1215.459,242.080,-61.179,-177.072,6.515,148.327
C05138=1215.463,241.831,-61.153,-177.075,6.513,148.327
C05139=1215.468,241.583,-61.127,-177.077,6.511,148.327
C05140=1215.473,241.334,-61.100,-177.080,6.508,148.328
C05141=1215.477,241.085,-61.075,-177.083,6.507,148.328
C05142=1215.481,240.837,-61.049,-177.085,6.504,148.328
C05143=1215.486,240.588,-61.022,-177.088,6.503,148.328
C05144=1215.490,240.339,-60.996,-177.090,6.501,148.329
C05145=1215.495,240.091,-60.971,-177.093,6.499,148.329
C05146=1215.499,239.842,-60.945,-177.095,6.497,148.329
C05147=1215.504,239.594,-60.918,-177.098,6.495,148.330
C05148=1215.508,239.345,-60.892,-177.100,6.493,148.330
C05149=1215.513,239.097,-60.867,-177.103,6.491,148.330
C05150=1215.517,238.848,-60.841,-177.105,6.489,148.330
C05151=1215.522,238.599,-60.815,-177.108,6.486,148.331
C05152=1215.526,238.350,-60.789,-177.111,6.484,148.331
C05153=1215.530,238.102,-60.762,-177.114,6.482,148.331
C05154=1215.535,237.854,-60.737,-177.116,6.480,148.331
C05155=1215.540,237.582,-60.709,-177.118,6.478,148.332
C05156=1215.545,237.310,-60.681,-177.121,6.477,148.332
C05157=1215.550,237.040,-60.653,-177.124,6.474,148.332
C05158=1215.555,236.767,-60.624,-177.127,6.472,148.332
C05159=1215.560,236.519,-60.599,-177.129,6.470,148.333
C05160=1215.564,236.270,-60.573,-177.132,6.468,148.333
C05161=1215.568,236.022,-60.547,-177.134,6.466,148.333
C05162=1215.573,235.773,-60.521,-177.137,6.464,148.334
C05163=1215.577,235.525,-60.496,-177.140,6.462,148.334
C05164=1215.582,235.276,-60.470,-177.143,6.460,148.334
C05165=1215.587,235.027,-60.444,-177.145,6.458,148.334
C05166=1215.591,234.779,-60.418,-177.147,6.456,148.335
C05167=1215.596,234.530,-60.393,-177.150,6.454,148.335
C05168=1215.600,234.281,-60.367,-177.153,6.452,148.335
C05169=1215.604,234.032,-60.341,-177.155,6.450,148.335
C05170=1215.609,233.784,-60.316,-177.157,6.448,148.336
C05171=1215.613,233.535,-60.290,-177.160,6.446,148.336
C05172=1215.617,233.287,-60.264,-177.163,6.444,148.336
C05173=1215.622,233.039,-60.239,-177.165,6.442,148.337
C05174=1215.626,232.790,-60.213,-177.167,6.440,148.337
C05175=1215.631,232.541,-60.187,-177.170,6.438,148.337
C05176=1215.635,232.293,-60.162,-177.173,6.436,148.337
C05177=1215.640,232.044,-60.136,-177.175,6.435,148.338
C05178=1215.644,231.795,-60.111,-177.178,6.433,148.338
C05179=1215.649,231.546,-60.086,-177.180,6.431,148.338
C05180=1215.653,231.298,-60.060,-177.183,6.429,148.338
C05181=1215.658,231.050,-60.035,-177.186,6.426,148.339
C05182=1215.662,230.801,-60.009,-177.189,6.424,148.339
C05183=1215.666,230.552,-59.983,-177.191,6.422,148.339
C05184=1215.672,230.303,-59.959,-177.193,6.420,148.339
C05185=1215.676,230.054,-59.933,-177.196,6.418,148.340
C05186=1215.680,229.806,-59.907,-177.199,6.416,148.340
C05187=1215.685,229.558,-59.882,-177.201,6.415,148.340
C05188=1215.689,229.308,-59.857,-177.204,6.413,148.341
C05189=1215.694,229.060,-59.831,-177.206,6.411,148.341
C05190=1215.698,228.811,-59.806,-177.209,6.409,148.341
C05191=1215.703,228.562,-59.780,-177.211,6.407,148.341
C05192=1215.708,228.314,-59.755,-177.214,6.405,148.342
C05193=1215.712,228.065,-59.729,-177.216,6.403,148.342
C05194=1215.717,227.817,-59.704,-177.219,6.401,148.342
C05195=1215.721,227.567,-59.679,-177.221,6.399,148.343
C05196=1215.726,227.319,-59.654,-177.224,6.397,148.343
C05197=1215.730,227.071,-59.628,-177.226,6.395,148.343
C05198=1215.734,226.821,-59.603,-177.229,6.393,148.344
C05199=1215.739,226.573,-59.578,-177.232,6.392,148.344
C05200=1215.743,226.324,-59.552,-177.234,6.390,148.344
C05201=1215.748,226.076,-59.528,-177.237,6.388,148.344
C05202=1215.753,225.827,-59.502,-177.239,6.386,148.345
C05203=1215.758,225.578,-59.477,-177.242,6.384,148.345
C05204=1215.761,225.330,-59.452,-177.244,6.382,148.345
C05205=1215.766,225.081,-59.427,-177.247,6.380,148.346
C05206=1215.771,224.832,-59.402,-177.250,6.378,148.346
C05207=1215.775,224.584,-59.376,-177.252,6.376,148.346
C05208=1215.780,224.335,-59.351,-177.254,6.374,148.346
C05209=1215.785,224.087,-59.326,-177.257,6.372,148.347
C05210=1215.789,223.837,-59.301,-177.260,6.371,148.347
C05211=1215.793,223.589,-59.276,-177.262,6.369,148.347
C05212=1215.798,223.340,-59.251,-177.265,6.367,148.348
C05213=1215.803,223.092,-59.225,-177.268,6.365,148.348
C05214=1215.807,222.843,-59.201,-177.270,6.363,148.348
C05215=1215.812,222.594,-59.176,-177.272,6.361,148.348
C05216=1215.816,222.345,-59.151,-177.275,6.359,148.349
C05217=1215.821,222.096,-59.126,-177.278,6.357,148.349
C05218=1215.825,221.848,-59.101,-177.280,6.355,148.349
C05219=1215.830,221.599,-59.076,-177.283,6.354,148.350
C05220=1215.834,221.350,-59.050,-177.286,6.352,148.350
C05221=1215.838,221.102,-59.026,-177.288,6.350,148.350
C05222=1215.843,220.853,-59.001,-177.291,6.348,148.351
C05223=1215.848,220.604,-58.976,-177.293,6.346,148.351
C05224=1215.853,220.356,-58.951,-177.296,6.344,148.351
C05225=1215.857,220.107,-58.927,-177.298,6.342,148.351
C05226=1215.861,219.858,-58.901,-177.301,6.340,148.352
C05227=1215.866,219.609,-58.876,-177.304,6.339,148.352
C05228=1215.870,219.361,-58.852,-177.306,6.337,148.352
C05229=1215.875,219.112,-58.827,-177.309,6.335,148.353
C05230=1215.879,218.863,-58.802,-177.311,6.333,148.353
C05231=1215.884,218.615,-58.778,-177.314,6.331,148.353
C05232=1215.889,218.365,-58.753,-177.317,6.329,148.354
C05233=1215.893,218.117,-58.728,-177.319,6.327,148.354
C05234=1215.897,217.868,-58.703,-177.321,6.325,148.354
C05235=1215.902,217.619,-58.678,-177.324,6.323,148.355
C05236=1215.907,217.371,-58.654,-177.327,6.322,148.355
C05237=1215.911,217.122,-58.628,-177.329,6.320,148.355
C05238=1215.915,216.874,-58.604,-177.332,6.318,148.356
C05239=1215.920,216.624,-58.579,-177.335,6.316,148.356
C05240=1215.924,216.376,-58.555,-177.337,6.314,148.356
C05241=1215.929,216.127,-58.531,-177.340,6.312,148.357
C05242=1215.934,215.878,-58.506,-177.343,6.310,148.357
C05243=1215.938,215.630,-58.481,-177.345,6.309,148.357
C05244=1215.943,215.381,-58.456,-177.348,6.307,148.358
C05245=1215.947,215.132,-58.432,-177.350,6.305,148.358
C05246=1215.952,214.883,-58.407,-177.353,6.303,148.358
C05247=1215.957,214.635,-58.383,-177.356,6.301,148.359
C05248=1215.961,214.386,-58.358,-177.358,6.299,148.359
C05249=1215.965,214.137,-58.334,-177.361,6.297,148.359
C05250=1215.971,213.888,-58.309,-177.363,6.295,148.359
C05251=1215.974,213.639,-58.285,-177.366,6.294,148.360
C05252=1215.979,213.391,-58.260,-177.368,6.292,148.360
C05253=1215.984,213.142,-58.236,-177.371,6.290,148.360
C05254=1215.988,212.893,-58.211,-177.374,6.288,148.361
C05255=1215.993,212.644,-58.187,-177.376,6.287,148.361
C05256=1215.998,212.396,-58.162,-177.378,6.285,148.361
C05257=1216.002,212.146,-58.138,-177.381,6.283,148.362
C05258=1216.006,211.898,-58.114,-177.384,6.281,148.362
C05259=1216.011,211.628,-58.087,-177.387,6.279,148.362
C05260=1216.016,211.358,-58.060,-177.390,6.277,148.363
C05261=1216.022,211.088,-58.034,-177.392,6.275,148.363
C05262=1216.026,210.816,-58.007,-177.395,6.273,148.363
C05263=1216.031,210.568,-57.983,-177.397,6.271,148.364
C05264=1216.035,210.319,-57.959,-177.400,6.270,148.364
C05265=1216.040,210.071,-57.934,-177.403,6.268,148.364
C05266=1216.044,209.821,-57.910,-177.405,6.266,148.365
C05267=1216.049,209.573,-57.885,-177.408,6.264,148.365
C05268=1216.054,209.324,-57.861,-177.411,6.262,148.365
C05269=1216.058,209.076,-57.837,-177.413,6.260,148.366
C05270=1216.063,208.826,-57.813,-177.416,6.258,148.366
C05271=1216.067,208.577,-57.789,-177.419,6.257,148.366
C05272=1216.072,208.329,-57.765,-177.421,6.256,148.367
C05273=1216.077,208.080,-57.740,-177.423,6.254,148.367
C05274=1216.081,207.832,-57.716,-177.426,6.252,148.367
C05275=1216.085,207.582,-57.692,-177.429,6.250,148.368
C05276=1216.090,207.333,-57.667,-177.431,6.248,148.368
C05277=1216.095,207.085,-57.643,-177.434,6.246,148.368
C05278=1216.099,206.837,-57.619,-177.436,6.245,148.369
C05279=1216.104,206.588,-57.595,-177.439,6.243,148.369
C05280=1216.108,206.338,-57.571,-177.442,6.241,148.369
C05281=1216.113,206.090,-57.547,-177.444,6.239,148.370
C05282=1216.117,205.841,-57.523,-177.447,6.237,148.370
C05283=1216.123,205.592,-57.499,-177.450,6.235,148.370
C05284=1216.127,205.344,-57.475,-177.452,6.234,148.371
C05285=1216.131,205.094,-57.450,-177.454,6.233,148.371
C05286=1216.136,204.845,-57.427,-177.457,6.231,148.371
C05287=1216.140,204.597,-57.403,-177.460,6.229,148.372
C05288=1216.145,204.348,-57.378,-177.462,6.227,148.372
C05289=1216.150,204.099,-57.355,-177.465,6.225,148.372
C05290=1216.154,203.851,-57.331,-177.468,6.223,148.373
C05291=1216.159,203.602,-57.307,-177.470,6.221,148.373
C05292=1216.163,203.353,-57.283,-177.473,6.220,148.373
C05293=1216.168,203.104,-57.258,-177.475,6.219,148.374
C05294=1216.173,202.855,-57.235,-177.478,6.217,148.374
C05295=1216.177,202.606,-57.211,-177.480,6.215,148.375
C05296=1216.181,202.358,-57.187,-177.483,6.213,148.375
C05297=1216.186,202.109,-57.163,-177.486,6.211,148.375
C05298=1216.190,201.861,-57.139,-177.488,6.209,148.376
C05299=1216.196,201.611,-57.115,-177.491,6.208,148.376
C05300=1216.200,201.363,-57.091,-177.493,6.206,148.376
C05301=1216.204,201.113,-57.068,-177.496,6.204,148.377
C05302=1216.209,200.865,-57.044,-177.498,6.203,148.377
C05303=1216.213,200.616,-57.020,-177.501,6.201,148.377
C05304=1216.218,200.367,-56.996,-177.503,6.199,148.378
C05305=1216.223,200.118,-56.973,-177.506,6.197,148.378
C05306=1216.227,199.870,-56.949,-177.509,6.196,148.378
C05307=1216.232,199.621,-56.925,-177.512,6.194,148.379
C05308=1216.236,199.372,-56.902,-177.515,6.192,148.379
C05309=1216.241,199.123,-56.878,-177.517,6.190,148.380
C05310=1216.246,198.874,-56.854,-177.519,6.189,148.380
C05311=1216.251,198.626,-56.830,-177.522,6.188,148.380
C05312=1216.255,198.377,-56.806,-177.525,6.186,148.381
C05313=1216.260,198.128,-56.783,-177.527,6.184,148.381
C05314=1216.264,197.879,-56.759,-177.530,6.182,148.381
C05315=1216.269,197.630,-56.736,-177.533,6.180,148.382
C05316=1216.273,197.382,-56.712,-177.535,6.179,148.382
C05317=1216.278,197.133,-56.688,-177.537,6.177,148.382
C05318=1216.283,196.884,-56.665,-177.540,6.176,148.383
C05319=1216.288,196.635,-56.642,-177.543,6.174,148.383
C05320=1216.292,196.386,-56.617,-177.545,6.172,148.383
C05321=1216.297,196.137,-56.594,-177.548,6.170,148.384
C05322=1216.301,195.888,-56.571,-177.550,6.168,148.384
C05323=1216.306,195.640,-56.547,-177.553,6.167,148.385
C05324=1216.310,195.391,-56.523,-177.555,6.165,148.385
C05325=1216.315,195.142,-56.500,-177.558,6.163,148.385
C05326=1216.319,194.893,-56.477,-177.560,6.162,148.386
C05327=1216.323,194.645,-56.453,-177.564,6.160,148.386
C05328=1216.328,194.395,-56.430,-177.566,6.158,148.386
C05329=1216.333,194.146,-56.406,-177.568,6.157,148.387
C05330=1216.338,193.897,-56.383,-177.571,6.155,148.387
C05331=1216.342,193.648,-56.360,-177.574,6.154,148.388
C05332=1216.347,193.400,-56.336,-177.576,6.152,148.388
C05333=1216.351,193.151,-56.312,-177.579,6.150,148.388
C05334=1216.356,192.902,-56.289,-177.582,6.148,148.389
C05335=1216.361,192.653,-56.266,-177.584,6.147,148.389
C05336=1216.365,192.404,-56.242,-177.586,6.145,148.389
C05337=1216.369,192.155,-56.219,-177.589,6.143,148.390
C05338=1216.374,191.906,-56.196,-177.592,6.142,148.390
C05339=1216.379,191.658,-56.172,-177.594,6.140,148.390
C05340=1216.383,191.409,-56.149,-177.597,6.139,148.391
C05341=1216.388,191.160,-56.125,-177.600,6.137,148.391
C05342=1216.393,190.911,-56.102,-177.602,6.135,148.392
C05343=1216.398,190.662,-56.079,-177.605,6.134,148.392
C05344=1216.402,190.414,-56.056,-177.607,6.132,148.392
C05345=1216.407,190.164,-56.033,-177.610,6.131,148.393
C05346=1216.411,189.915,-56.009,-177.612,6.129,148.393
C05347=1216.416,189.666,-55.986,-177.615,6.127,148.393
C05348=1216.421,189.417,-55.963,-177.617,6.125,148.394
C05349=1216.425,189.169,-55.940,-177.620,6.123,148.394
C05350=1216.429,188.920,-55.917,-177.623,6.123,148.395
C05351=1216.435,188.671,-55.894,-177.625,6.121,148.395
C05352=1216.439,188.422,-55.870,-177.628,6.119,148.395
C05353=1216.443,188.174,-55.847,-177.631,6.117,148.396
C05354=1216.448,187.925,-55.824,-177.633,6.116,148.396
C05355=1216.453,187.675,-55.801,-177.635,6.115,148.396
C05356=1216.457,187.426,-55.777,-177.638,6.113,148.397
C05357=1216.461,187.178,-55.755,-177.641,6.111,148.397
C05358=1216.467,186.929,-55.732,-177.643,6.109,148.398
C05359=1216.472,186.680,-55.709,-177.646,6.108,148.398
C05360=1216.476,186.431,-55.686,-177.649,6.107,148.398
C05361=1216.480,186.182,-55.663,-177.651,6.105,148.399
C05362=1216.485,185.933,-55.640,-177.654,6.103,148.399
C05363=1216.490,185.663,-55.615,-177.657,6.101,148.400
C05364=1216.495,185.394,-55.590,-177.660,6.100,148.400
C05365=1216.500,185.124,-55.565,-177.662,6.098,148.400
C05366=1216.505,184.855,-55.541,-177.665,6.096,148.401
C05367=1216.510,184.605,-55.517,-177.668,6.094,148.401
C05368=1216.515,184.357,-55.494,-177.670,6.093,148.402
C05369=1216.519,184.108,-55.471,-177.673,6.092,148.402
C05370=1216.524,183.859,-55.449,-177.676,6.090,148.402
C05371=1216.528,183.610,-55.426,-177.678,6.088,148.403
C05372=1216.532,183.361,-55.403,-177.680,6.087,148.403
C05373=1216.538,183.113,-55.380,-177.683,6.085,148.404
C05374=1216.542,182.863,-55.358,-177.686,6.083,148.404
C05375=1216.547,182.614,-55.334,-177.688,6.081,148.404
C05376=1216.551,182.366,-55.312,-177.691,6.081,148.405
C05377=1216.556,182.117,-55.289,-177.693,6.079,148.405
C05378=1216.561,181.868,-55.266,-177.696,6.077,148.406
C05379=1216.565,181.619,-55.243,-177.699,6.075,148.406
C05380=1216.570,181.370,-55.220,-177.701,6.074,148.406
C05381=1216.575,181.121,-55.198,-177.703,6.072,148.407
C05382=1216.579,180.872,-55.175,-177.706,6.071,148.407
C05383=1216.583,180.623,-55.152,-177.709,6.069,148.408
C05384=1216.588,180.374,-55.129,-177.711,6.068,148.408
C05385=1216.593,180.126,-55.107,-177.714,6.066,148.408
C05386=1216.598,179.876,-55.084,-177.717,6.065,148.409
C05387=1216.602,179.627,-55.062,-177.719,6.063,148.409
C05388=1216.607,179.379,-55.039,-177.721,6.062,148.409
C05389=1216.611,179.130,-55.016,-177.725,6.060,148.410
C05390=1216.616,178.881,-54.993,-177.727,6.058,148.410
C05391=1216.620,178.631,-54.971,-177.730,6.057,148.411
C05392=1216.626,178.383,-54.948,-177.732,6.056,148.411
C05393=1216.630,178.134,-54.926,-177.735,6.054,148.411
C05394=1216.635,177.885,-54.903,-177.737,6.052,148.412
C05395=1216.639,177.636,-54.881,-177.740,6.051,148.412
C05396=1216.644,177.387,-54.858,-177.743,6.049,148.413
C05397=1216.648,177.138,-54.836,-177.745,6.048,148.413
C05398=1216.654,176.889,-54.813,-177.748,6.046,148.414
C05399=1216.658,176.640,-54.791,-177.750,6.045,148.414
C05400=1216.662,176.391,-54.768,-177.753,6.043,148.414
C05401=1216.668,176.142,-54.745,-177.756,6.041,148.415
C05402=1216.671,175.894,-54.723,-177.758,6.040,148.415
C05403=1216.676,175.644,-54.700,-177.760,6.039,148.416
C05404=1216.681,175.396,-54.678,-177.763,6.037,148.416
C05405=1216.685,175.147,-54.656,-177.766,6.035,148.416
C05406=1216.691,174.898,-54.633,-177.768,6.034,148.417
C05407=1216.695,174.649,-54.611,-177.771,6.033,148.417
C05408=1216.700,174.399,-54.588,-177.774,6.031,148.418
C05409=1216.705,174.151,-54.566,-177.776,6.030,148.418
C05410=1216.709,173.902,-54.544,-177.778,6.028,148.418
C05411=1216.714,173.653,-54.521,-177.782,6.026,148.419
C05412=1216.718,173.404,-54.498,-177.784,6.025,148.419
C05413=1216.723,173.155,-54.476,-177.786,6.024,148.420
C05414=1216.728,172.906,-54.454,-177.789,6.022,148.420
C05415=1216.732,172.657,-54.432,-177.792,6.020,148.420
C05416=1216.737,172.409,-54.410,-177.794,6.019,148.421
C05417=1216.741,172.159,-54.388,-177.797,6.017,148.421
C05418=1216.746,171.910,-54.365,-177.800,6.016,148.422
C05419=1216.751,171.662,-54.343,-177.802,6.015,148.422
C05420=1216.755,171.412,-54.321,-177.805,6.013,148.423
C05421=1216.761,171.163,-54.298,-177.807,6.011,148.423
C05422=1216.765,170.914,-54.276,-177.810,6.010,148.423
C05423=1216.770,170.666,-54.254,-177.812,6.009,148.424
C05424=1216.774,170.417,-54.232,-177.815,6.007,148.424
C05425=1216.779,170.168,-54.210,-177.817,6.006,148.425
C05426=1216.784,169.918,-54.187,-177.820,6.004,148.425
C05427=1216.788,169.669,-54.165,-177.823,6.002,148.426
C05428=1216.793,169.421,-54.143,-177.825,6.001,148.426
C05429=1216.798,169.171,-54.120,-177.828,6.000,148.427
C05430=1216.802,168.923,-54.099,-177.831,5.998,148.427
C05431=1216.807,168.673,-54.077,-177.833,5.997,148.427
C05432=1216.812,168.425,-54.055,-177.835,5.995,148.428
C05433=1216.816,168.175,-54.033,-177.838,5.994,148.428
C05434=1216.821,167.926,-54.011,-177.841,5.993,148.429
C05435=1216.826,167.677,-53.989,-177.843,5.991,148.429
C05436=1216.830,167.429,-53.966,-177.846,5.989,148.429
C05437=1216.835,167.180,-53.944,-177.848,5.988,148.430
C05438=1216.839,166.931,-53.922,-177.851,5.987,148.430
C05439=1216.844,166.682,-53.900,-177.854,5.985,148.431
C05440=1216.849,166.433,-53.878,-177.856,5.984,148.431
C05441=1216.854,166.183,-53.856,-177.859,5.982,148.431
C05442=1216.858,165.935,-53.834,-177.862,5.981,148.432
C05443=1216.863,165.685,-53.812,-177.864,5.980,148.432
C05444=1216.868,165.437,-53.791,-177.867,5.978,148.433
C05445=1216.872,165.188,-53.769,-177.869,5.976,148.433
C05446=1216.877,164.939,-53.747,-177.872,5.975,148.434
C05447=1216.882,164.690,-53.725,-177.875,5.974,148.434
C05448=1216.886,164.441,-53.703,-177.877,5.973,148.435
C05449=1216.891,164.192,-53.682,-177.879,5.971,148.435
C05450=1216.896,163.942,-53.659,-177.882,5.969,148.435
C05451=1216.901,163.694,-53.637,-177.885,5.968,148.436
C05452=1216.905,163.445,-53.615,-177.887,5.967,148.436
C05453=1216.910,163.196,-53.593,-177.890,5.965,148.437
C05454=1216.915,162.947,-53.572,-177.892,5.964,148.437
C05455=1216.919,162.697,-53.550,-177.895,5.962,148.438
C05456=1216.924,162.449,-53.529,-177.897,5.961,148.438
C05457=1216.928,162.199,-53.507,-177.900,5.960,148.439
C05458=1216.933,161.951,-53.485,-177.903,5.958,148.439
C05459=1216.938,161.702,-53.463,-177.905,5.957,148.439
C05460=1216.942,161.453,-53.441,-177.908,5.955,148.440
C05461=1216.947,161.204,-53.420,-177.911,5.954,148.440
C05462=1216.952,160.954,-53.398,-177.913,5.953,148.441
C05463=1216.957,160.705,-53.377,-177.916,5.951,148.441
C05464=1216.961,160.457,-53.355,-177.918,5.950,148.441
C05465=1216.966,160.207,-53.333,-177.921,5.948,148.442
C05466=1216.971,159.959,-53.311,-177.924,5.947,148.442
C05467=1216.975,159.690,-53.288,-177.926,5.946,148.443
C05468=1216.981,159.420,-53.265,-177.929,5.944,148.443
C05469=1216.985,159.152,-53.242,-177.932,5.942,148.444
C05470=1216.991,158.883,-53.218,-177.935,5.941,148.444
